LIN {X 0,Y 269.087,Z 444.894,A -85,B 0,C 180,E1 -18604.681,E2 -18604.681} C_VEL
LIN {X 0,Y 267.627,Z 456.093,A -85,B 0,C 180,E1 -18605.777,E2 -18605.777} C_VEL
LIN {X 0,Y 265.719,Z 467.668,A -85,B 0,C 180,E1 -18607.245,E2 -18607.245} C_VEL
LIN {X 0,Y 263.911,Z 478.137,A -85,B 0,C 180,E1 -18608.962,E2 -18608.962} C_VEL
LIN {X 0,Y 262.001,Z 487.303,A -85,B 0,C 180,E1 -18610.818,E2 -18610.818} C_VEL
LIN {X 0,Y 259.893,Z 496.269,A -85,B 0,C 180,E1 -18613.102,E2 -18613.102} C_VEL
LIN {X 0,Y 258.271,Z 503.459,A -85,B 0,C 180,E1 -18615.423,E2 -18615.423} C_VEL
LIN {X 0,Y 256.682,Z 510.056,A -85,B 0,C 180,E1 -18618.152,E2 -18618.152} C_VEL
LIN {X 0,Y 255.709,Z 514.379,A -85,B 0,C 180,E1 -18620.51,E2 -18620.51} C_VEL
LIN {X 0,Y 255.059,Z 517.472,A -85,B 0,C 180,E1 -18622.731,E2 -18622.731} C_VEL
LIN {X 0,Y 254.598,Z 519.914,A -85,B 0,C 180,E1 -18625.251,E2 -18625.251} C_VEL
LIN {X 0,Y 254.212,Z 521.518,A -85,B 0,C 180,E1 -18628.417,E2 -18628.417} C_VEL
LIN {X 0,Y 254.18,Z 521.749,A -85,B 0,C 180,E1 -18630.002,E2 -18630.002} C_VEL
LIN {X 0,Y 254.364,Z 520.966,A -85,B 0,C 180,E1 -18633.169,E2 -18633.169} C_VEL
LIN {X 0,Y 254.595,Z 519.999,A -85,B 0,C 180,E1 -18634.752,E2 -18634.752} C_VEL
LIN {X 0,Y 255.074,Z 517.58,A -85,B 0,C 180,E1 -18637.295,E2 -18637.295} C_VEL
LIN {X 0,Y 255.634,Z 514.567,A -85,B 0,C 180,E1 -18639.496,E2 -18639.496} C_VEL
LIN {X 0,Y 256.622,Z 510.299,A -85,B 0,C 180,E1 -18641.854,E2 -18641.854} C_VEL
LIN {X 0,Y 257.962,Z 504.844,A -85,B 0,C 180,E1 -18644.195,E2 -18644.195} C_VEL
LIN {X 0,Y 259.535,Z 497.997,A -85,B 0,C 180,E1 -18646.52,E2 -18646.52} C_VEL
LIN {X 0,Y 261.635,Z 489.404,A -85,B 0,C 180,E1 -18648.806,E2 -18648.806} C_VEL
LIN {X 0,Y 263.444,Z 480.947,A -85,B 0,C 180,E1 -18650.627,E2 -18650.627} C_VEL
LIN {X 0,Y 265.212,Z 470.915,A -85,B 0,C 180,E1 -18652.393,E2 -18652.393} C_VEL
LIN {X 0,Y 267.064,Z 460.167,A -85,B 0,C 180,E1 -18653.868,E2 -18653.868} C_VEL
LIN {X 0,Y 268.762,Z 448.198,A -85,B 0,C 180,E1 -18655.148,E2 -18655.148} C_VEL
LIN {X 0,Y 270.109,Z 435.553,A -85,B 0,C 180,E1 -18656.15,E2 -18656.15} C_VEL
LIN {X 0,Y 271.18,Z 422.049,A -85,B 0,C 180,E1 -18656.868,E2 -18656.868} C_VEL
LIN {X 0,Y 271.846,Z 405.573,A -85,B 0,C 180,E1 -18657.369,E2 -18657.369} C_VEL
LIN {X 0,Y 273.565,Z 348.69,A -85,B 0,C 180,E1 -18658.847,E2 -18658.847} C_VEL
LIN {X 0,Y 265.912,Z 332.327,A -85,B 0,C 180,E1 -18660.269,E2 -18660.269} C_VEL
LIN {X 0,Y 257.649,Z 317.178,A -85,B 0,C 180,E1 -18661.844,E2 -18661.844} C_VEL
LIN {X 0,Y 256.315,Z 314.678,A -85,B 0,C 180,E1 -18662.112,E2 -18662.112} C_VEL
LIN {X 0,Y 256.105,Z 313.584,A -85,B 0,C 180,E1 -18662.211,E2 -18662.211} C_VEL
LIN {X 0,Y 256.126,Z 313.582,A -85,B 0,C 180,E1 -18665.188,E2 -18665.188} C_VEL
LIN {X 0,Y 256.097,Z 313.587,A -85,B 0,C 180,E1 -18669.139,E2 -18669.139} C_VEL
LIN {X 0,Y 256.078,Z 313.582,A -85,B 0,C 180,E1 -18673.326,E2 -18673.326} C_VEL
LIN {X 0,Y 256.079,Z 313.572,A -85,B 0,C 180,E1 -18677.819,E2 -18677.819} C_VEL
LIN {X 0,Y 256.077,Z 313.589,A -85,B 0,C 180,E1 -18680.859,E2 -18680.859} C_VEL
LIN {X 0,Y 256.135,Z 313.573,A -85,B 0,C 180,E1 -18682.868,E2 -18682.868} C_VEL
LIN {X 0,Y 256.073,Z 313.588,A -85,B 0,C 180,E1 -18686.708,E2 -18686.708} C_VEL
LIN {X 0,Y 256.119,Z 313.574,A -85,B 0,C 180,E1 -18690.401,E2 -18690.401} C_VEL
LIN {X 0,Y 256.217,Z 313.561,A -85,B 0,C 180,E1 -18694.995,E2 -18694.995} C_VEL
LIN {X 0,Y 263.531,Z 341.555,A -85,B 0,C 180,E1 -18696.573,E2 -18696.573} C_VEL
LIN {X 0,Y 260.281,Z 420.849,A -85,B 0,C 180,E1 -18700.068,E2 -18700.068} C_VEL
LIN {X 0,Y 260.015,Z 427.794,A -85,B 0,C 180,E1 -18700.495,E2 -18700.495} C_VEL
LIN {X 0,Y 258.964,Z 433.354,A -85,B 0,C 180,E1 -18700.879,E2 -18700.879} C_VEL
LIN {X 0,Y 255.487,Z 442.099,A -85,B 0,C 180,E1 -18701.589,E2 -18701.589} C_VEL
LIN {X 0,Y 252.06,Z 450.609,A -85,B 0,C 180,E1 -18702.446,E2 -18702.446} C_VEL
LIN {X 0,Y 251.094,Z 455.788,A -85,B 0,C 180,E1 -18703.062,E2 -18703.062} C_VEL
LIN {X 0,Y 250.361,Z 465.042,A -85,B 0,C 180,E1 -18704.324,E2 -18704.324} C_VEL
LIN {X 0,Y 249.484,Z 476.008,A -85,B 0,C 180,E1 -18706.146,E2 -18706.146} C_VEL
LIN {X 0,Y 248.674,Z 486,A -85,B 0,C 180,E1 -18708.176,E2 -18708.176} C_VEL
LIN {X 0,Y 248.087,Z 494.293,A -85,B 0,C 180,E1 -18710.214,E2 -18710.214} C_VEL
LIN {X 0,Y 247.557,Z 502.409,A -85,B 0,C 180,E1 -18712.66,E2 -18712.66} C_VEL
LIN {X 0,Y 247.21,Z 508.939,A -85,B 0,C 180,E1 -18715.107,E2 -18715.107} C_VEL
LIN {X 0,Y 247.148,Z 514.155,A -85,B 0,C 180,E1 -18717.555,E2 -18717.555} C_VEL
LIN {X 0,Y 247.07,Z 518.167,A -85,B 0,C 180,E1 -18720,E2 -18720} C_VEL
LIN {X 0,Y 247.189,Z 520.272,A -85,B 0,C 180,E1 -18721.629,E2 -18721.629} C_VEL
LIN {X 0,Y 247.43,Z 521.895,A -85,B 0,C 180,E1 -18723.257,E2 -18723.257} C_VEL
LIN {X 0,Y 247.715,Z 523.106,A -85,B 0,C 180,E1 -18724.883,E2 -18724.883} C_VEL
LIN {X 0,Y 248.077,Z 523.926,A -85,B 0,C 180,E1 -18726.507,E2 -18726.507} C_VEL
LIN {X 0,Y 249.255,Z 524.369,A -85,B 0,C 180,E1 -18729.29,E2 -18729.29} C_VEL
LIN {X 0,Y 250.523,Z 523.882,A -85,B 0,C 180,E1 -18731.325,E2 -18731.325} C_VEL
LIN {X 0,Y 252.837,Z 521.893,A -85,B 0,C 180,E1 -18734.487,E2 -18734.487} C_VEL
LIN {X 0,Y 255.28,Z 519.262,A -85,B 0,C 180,E1 -18736.802,E2 -18736.802} C_VEL
LIN {X 0,Y 258.013,Z 515.67,A -85,B 0,C 180,E1 -18739.079,E2 -18739.079} C_VEL
LIN {X 0,Y 261.191,Z 511.028,A -85,B 0,C 180,E1 -18741.3,E2 -18741.3} C_VEL
LIN {X 0,Y 265.442,Z 504.122,A -85,B 0,C 180,E1 -18743.814,E2 -18743.814} C_VEL
LIN {X 0,Y 270.342,Z 495.356,A -85,B 0,C 180,E1 -18746.228,E2 -18746.228} C_VEL
LIN {X 0,Y 274.943,Z 485.994,A -85,B 0,C 180,E1 -18748.222,E2 -18748.222} C_VEL
LIN {X 0,Y 279.433,Z 475.658,A -85,B 0,C 180,E1 -18749.992,E2 -18749.992} C_VEL
LIN {X 0,Y 283.883,Z 464.048,A -85,B 0,C 180,E1 -18751.533,E2 -18751.533} C_VEL
LIN {X 0,Y 288.003,Z 451.271,A -85,B 0,C 180,E1 -18752.885,E2 -18752.885} C_VEL
LIN {X 0,Y 291.73,Z 437.57,A -85,B 0,C 180,E1 -18753.959,E2 -18753.959} C_VEL
LIN {X 0,Y 294.428,Z 424.942,A -85,B 0,C 180,E1 -18754.691,E2 -18754.691} C_VEL
LIN {X 0,Y 301.418,Z 387.209,A -85,B 0,C 180,E1 -18756.436,E2 -18756.436} C_VEL
LIN {X 0,Y 299.691,Z 383.358,A -85,B 0,C 180,E1 -18758.133,E2 -18758.133} C_VEL
LIN {X 0,Y 298.164,Z 380.681,A -85,B 0,C 180,E1 -18759.997,E2 -18759.997} C_VEL
LIN {X 0,Y 296.756,Z 378.932,A -85,B 0,C 180,E1 -18762.762,E2 -18762.762} C_VEL
LIN {X 0,Y 296.466,Z 379.001,A -85,B 0,C 180,E1 -18764.984,E2 -18764.984} C_VEL
LIN {X 0,Y 296.557,Z 380.147,A -85,B 0,C 180,E1 -18766.453,E2 -18766.453} C_VEL
LIN {X 0,Y 297.703,Z 384.492,A -85,B 0,C 180,E1 -18769.469,E2 -18769.469} C_VEL
LIN {X 0,Y 299.157,Z 389.614,A -85,B 0,C 180,E1 -18771.566,E2 -18771.566} C_VEL
LIN {X 0,Y 300.305,Z 394.278,A -85,B 0,C 180,E1 -18772.933,E2 -18772.933} C_VEL
LIN {X 0,Y 300.019,Z 397.921,A -85,B 0,C 180,E1 -18773.303,E2 -18773.303} C_VEL
LIN {X 0,Y 292.072,Z 440.822,A -85,B 0,C 180,E1 -18775.25,E2 -18775.25} C_VEL
LIN {X 0,Y 288.407,Z 455.283,A -85,B 0,C 180,E1 -18776.121,E2 -18776.121} C_VEL
LIN {X 0,Y 284.066,Z 469.15,A -85,B 0,C 180,E1 -18777.233,E2 -18777.233} C_VEL
LIN {X 0,Y 279.463,Z 481.671,A -85,B 0,C 180,E1 -18778.544,E2 -18778.544} C_VEL
LIN {X 0,Y 274.353,Z 494.035,A -85,B 0,C 180,E1 -18780.242,E2 -18780.242} C_VEL
LIN {X 0,Y 269.677,Z 504.242,A -85,B 0,C 180,E1 -18782.023,E2 -18782.023} C_VEL
LIN {X 0,Y 265.145,Z 513.442,A -85,B 0,C 180,E1 -18784.063,E2 -18784.063} C_VEL
LIN {X 0,Y 261.091,Z 521.078,A -85,B 0,C 180,E1 -18786.185,E2 -18786.185} C_VEL
LIN {X 0,Y 257.423,Z 527.418,A -85,B 0,C 180,E1 -18788.367,E2 -18788.367} C_VEL
LIN {X 0,Y 254.576,Z 532.571,A -85,B 0,C 180,E1 -18790.652,E2 -18790.652} C_VEL
LIN {X 0,Y 252.113,Z 536.709,A -85,B 0,C 180,E1 -18792.979,E2 -18792.979} C_VEL
LIN {X 0,Y 250.025,Z 539.89,A -85,B 0,C 180,E1 -18795.344,E2 -18795.344} C_VEL
LIN {X 0,Y 248.241,Z 542.675,A -85,B 0,C 180,E1 -18798.568,E2 -18798.568} C_VEL
LIN {X 0,Y 247.251,Z 543.919,A -85,B 0,C 180,E1 -18801.828,E2 -18801.828} C_VEL
LIN {X 0,Y 247.04,Z 543.519,A -85,B 0,C 180,E1 -18805.102,E2 -18805.102} C_VEL
LIN {X 0,Y 247.072,Z 543.112,A -85,B 0,C 180,E1 -18806.357,E2 -18806.357} C_VEL
LIN {X 0,Y 247.095,Z 543.924,A -85,B 0,C 180,E1 -18808.369,E2 -18808.369} C_VEL
LIN {X 0,Y 247.224,Z 544.148,A -85,B 0,C 180,E1 -18809.998,E2 -18809.998} C_VEL
LIN {X 0,Y 247.139,Z 543.916,A -85,B 0,C 180,E1 -18811.628,E2 -18811.628} C_VEL
LIN {X 0,Y 247.041,Z 543.284,A -85,B 0,C 180,E1 -18813.26,E2 -18813.26} C_VEL
LIN {X 0,Y 246.951,Z 542.125,A -85,B 0,C 180,E1 -18815.08,E2 -18815.08} C_VEL
LIN {X 0,Y 247.192,Z 538.891,A -85,B 0,C 180,E1 -18818.171,E2 -18818.171} C_VEL
LIN {X 0,Y 247.681,Z 535.184,A -85,B 0,C 180,E1 -18820.627,E2 -18820.627} C_VEL
LIN {X 0,Y 248.483,Z 530.34,A -85,B 0,C 180,E1 -18823.076,E2 -18823.076} C_VEL
LIN {X 0,Y 249.928,Z 524.229,A -85,B 0,C 180,E1 -18825.492,E2 -18825.492} C_VEL
LIN {X 0,Y 251.653,Z 516.619,A -85,B 0,C 180,E1 -18827.889,E2 -18827.889} C_VEL
LIN {X 0,Y 253.266,Z 508.806,A -85,B 0,C 180,E1 -18829.871,E2 -18829.871} C_VEL
LIN {X 0,Y 255.341,Z 499.264,A -85,B 0,C 180,E1 -18831.811,E2 -18831.811} C_VEL
LIN {X 0,Y 257.545,Z 488.681,A -85,B 0,C 180,E1 -18833.52,E2 -18833.52} C_VEL
LIN {X 0,Y 259.374,Z 478.44,A -85,B 0,C 180,E1 -18834.832,E2 -18834.832} C_VEL
LIN {X 0,Y 261.082,Z 467.279,A -85,B 0,C 180,E1 -18835.938,E2 -18835.938} C_VEL
LIN {X 0,Y 262.693,Z 454.054,A -85,B 0,C 180,E1 -18836.89,E2 -18836.89} C_VEL
LIN {X 0,Y 263.806,Z 441.539,A -85,B 0,C 180,E1 -18837.483,E2 -18837.483} C_VEL
LIN {X 0,Y 265.629,Z 384.766,A -85,B 0,C 180,E1 -18839.024,E2 -18839.024} C_VEL
LIN {X 0,Y 261.716,Z 352.974,A -85,B 0,C 180,E1 -18840.477,E2 -18840.477} C_VEL
LIN {X 0,Y 260.479,Z 344.507,A -85,B 0,C 180,E1 -18840.9,E2 -18840.9} C_VEL
LIN {X 0,Y 253.85,Z 326.102,A -85,B 0,C 180,E1 -18842.391,E2 -18842.391} C_VEL
LIN {X 0,Y 250.812,Z 318.273,A -85,B 0,C 180,E1 -18843.122,E2 -18843.122} C_VEL
LIN {X 0,Y 249.277,Z 315.423,A -85,B 0,C 180,E1 -18843.494,E2 -18843.494} C_VEL
LIN {X 0,Y 249.094,Z 314.457,A -85,B 0,C 180,E1 -18843.611,E2 -18843.611} C_VEL
LIN {X 0,Y 249.044,Z 314.46,A -85,B 0,C 180,E1 -18847.8,E2 -18847.8} C_VEL
LIN {X 0,Y 249.001,Z 314.464,A -85,B 0,C 180,E1 -18850.477,E2 -18850.477} C_VEL
LIN {X 0,Y 248.978,Z 314.467,A -85,B 0,C 180,E1 -18854.882,E2 -18854.882} C_VEL
LIN {X 0,Y 248.978,Z 314.462,A -85,B 0,C 180,E1 -18857.355,E2 -18857.355} C_VEL
LIN {X 0,Y 249.014,Z 314.464,A -85,B 0,C 180,E1 -18862.206,E2 -18862.206} C_VEL
LIN {X 0,Y 249.035,Z 314.458,A -85,B 0,C 180,E1 -18865.638,E2 -18865.638} C_VEL
LIN {X 0,Y 248.986,Z 314.465,A -85,B 0,C 180,E1 -18869.464,E2 -18869.464} C_VEL
LIN {X 0,Y 249.007,Z 314.468,A -85,B 0,C 180,E1 -18873.155,E2 -18873.155} C_VEL
LIN {X 0,Y 249.003,Z 314.466,A -85,B 0,C 180,E1 -18876.725,E2 -18876.725} C_VEL
LIN {X 0,Y 249.05,Z 314.449,A -85,B 0,C 180,E1 -18880.207,E2 -18880.207} C_VEL
LIN {X 0,Y 249.15,Z 314.421,A -85,B 0,C 180,E1 -18883.616,E2 -18883.616} C_VEL
LIN {X 0,Y 249.203,Z 314.439,A -85,B 0,C 180,E1 -18886.961,E2 -18886.961} C_VEL
LIN {X 0,Y 249.375,Z 314.415,A -85,B 0,C 180,E1 -18890.522,E2 -18890.522} C_VEL
LIN {X 0,Y 249.416,Z 314.38,A -85,B 0,C 180,E1 -18893.528,E2 -18893.528} C_VEL
LIN {X 0,Y 249.649,Z 314.38,A -85,B 0,C 180,E1 -18898.387,E2 -18898.387} C_VEL
LIN {X 0,Y 249.65,Z 314.383,A -85,B 0,C 180,E1 -18901.613,E2 -18901.613} C_VEL
LIN {X 0,Y 249.405,Z 314.415,A -85,B 0,C 180,E1 -18906.662,E2 -18906.662} C_VEL
LIN {X 0,Y 249.335,Z 314.417,A -85,B 0,C 180,E1 -18909.737,E2 -18909.737} C_VEL
LIN {X 0,Y 249.168,Z 314.443,A -85,B 0,C 180,E1 -18914.706,E2 -18914.706} C_VEL
LIN {X 0,Y 249.101,Z 314.443,A -85,B 0,C 180,E1 -18918.08,E2 -18918.08} C_VEL
LIN {X 0,Y 249.073,Z 314.458,A -85,B 0,C 180,E1 -18921.52,E2 -18921.52} C_VEL
LIN {X 0,Y 249.097,Z 314.444,A -85,B 0,C 180,E1 -18925.47,E2 -18925.47} C_VEL
LIN {X 0,Y 249.034,Z 314.464,A -85,B 0,C 180,E1 -18928.977,E2 -18928.977} C_VEL
LIN {X 0,Y 249.021,Z 314.454,A -85,B 0,C 180,E1 -18932.427,E2 -18932.427} C_VEL
LIN {X 0,Y 249.042,Z 314.46,A -85,B 0,C 180,E1 -18936.344,E2 -18936.344} C_VEL
LIN {X 0,Y 249.001,Z 314.47,A -85,B 0,C 180,E1 -18940.479,E2 -18940.479} C_VEL
LIN {X 0,Y 248.989,Z 314.471,A -85,B 0,C 180,E1 -18944.883,E2 -18944.883} C_VEL
LIN {X 0,Y 249.012,Z 314.459,A -85,B 0,C 180,E1 -18947.364,E2 -18947.364} C_VEL
LIN {X 0,Y 249.041,Z 314.443,A -85,B 0,C 180,E1 -18952.202,E2 -18952.202} C_VEL
LIN {X 0,Y 249.054,Z 314.462,A -85,B 0,C 180,E1 -18955.643,E2 -18955.643} C_VEL
LIN {X 0,Y 249.043,Z 314.455,A -85,B 0,C 180,E1 -18956.913,E2 -18956.913} C_VEL
LIN {X 0,Y 250.179,Z 317.525,A -85,B 0,C 180,E1 -18957.232,E2 -18957.232} C_VEL
LIN {X 0,Y 255.198,Z 326.145,A -85,B 0,C 180,E1 -18958.242,E2 -18958.242} C_VEL
LIN {X 0,Y 263.451,Z 342.159,A -85,B 0,C 180,E1 -18959.855,E2 -18959.855} C_VEL
LIN {X 0,Y 267.251,Z 350.558,A -85,B 0,C 180,E1 -18960.587,E2 -18960.587} C_VEL
LIN {X 0,Y 264.927,Z 419.914,A -85,B 0,C 180,E1 -18962.464,E2 -18962.464} C_VEL
LIN {X 0,Y 263.995,Z 432.708,A -85,B 0,C 180,E1 -18963.093,E2 -18963.093} C_VEL
LIN {X 0,Y 262.699,Z 445.193,A -85,B 0,C 180,E1 -18964.02,E2 -18964.02} C_VEL
LIN {X 0,Y 261.185,Z 456.398,A -85,B 0,C 180,E1 -18965.14,E2 -18965.14} C_VEL
LIN {X 0,Y 259.426,Z 466.702,A -85,B 0,C 180,E1 -18966.45,E2 -18966.45} C_VEL
LIN {X 0,Y 257.635,Z 476.588,A -85,B 0,C 180,E1 -18968.046,E2 -18968.046} C_VEL
LIN {X 0,Y 255.736,Z 485.882,A -85,B 0,C 180,E1 -18969.91,E2 -18969.91} C_VEL
LIN {X 0,Y 253.438,Z 495.252,A -85,B 0,C 180,E1 -18972.241,E2 -18972.241} C_VEL
LIN {X 0,Y 251.682,Z 502.686,A -85,B 0,C 180,E1 -18974.618,E2 -18974.618} C_VEL
LIN {X 0,Y 250.172,Z 508.656,A -85,B 0,C 180,E1 -18977.014,E2 -18977.014} C_VEL
LIN {X 0,Y 249.021,Z 513.369,A -85,B 0,C 180,E1 -18979.431,E2 -18979.431} C_VEL
LIN {X 0,Y 248.22,Z 516.967,A -85,B 0,C 180,E1 -18981.863,E2 -18981.863} C_VEL
LIN {X 0,Y 247.791,Z 518.82,A -85,B 0,C 180,E1 -18983.487,E2 -18983.487} C_VEL
LIN {X 0,Y 247.531,Z 520.231,A -85,B 0,C 180,E1 -18985.115,E2 -18985.115} C_VEL
LIN {X 0,Y 247.305,Z 521.222,A -85,B 0,C 180,E1 -18986.743,E2 -18986.743} C_VEL
LIN {X 0,Y 247.105,Z 522.065,A -85,B 0,C 180,E1 -18990.002,E2 -18990.002} C_VEL
LIN {X 0,Y 247.304,Z 521.282,A -85,B 0,C 180,E1 -18993.26,E2 -18993.26} C_VEL
LIN {X 0,Y 247.528,Z 520.315,A -85,B 0,C 180,E1 -18994.888,E2 -18994.888} C_VEL
LIN {X 0,Y 248.006,Z 518.084,A -85,B 0,C 180,E1 -18997.327,E2 -18997.327} C_VEL
LIN {X 0,Y 248.648,Z 514.882,A -85,B 0,C 180,E1 -18999.766,E2 -18999.766} C_VEL
LIN {X 0,Y 249.691,Z 510.613,A -85,B 0,C 180,E1 -19002.188,E2 -19002.188} C_VEL
LIN {X 0,Y 251.08,Z 505.157,A -85,B 0,C 180,E1 -19004.593,E2 -19004.593} C_VEL
LIN {X 0,Y 252.742,Z 498.308,A -85,B 0,C 180,E1 -19006.978,E2 -19006.978} C_VEL
LIN {X 0,Y 254.939,Z 489.713,A -85,B 0,C 180,E1 -19009.319,E2 -19009.319} C_VEL
LIN {X 0,Y 257.036,Z 480.126,A -85,B 0,C 180,E1 -19011.414,E2 -19011.414} C_VEL
LIN {X 0,Y 258.928,Z 469.969,A -85,B 0,C 180,E1 -19013.178,E2 -19013.178} C_VEL
LIN {X 0,Y 260.859,Z 458.939,A -85,B 0,C 180,E1 -19014.684,E2 -19014.684} C_VEL
LIN {X 0,Y 262.494,Z 447.523,A -85,B 0,C 180,E1 -19015.898,E2 -19015.898} C_VEL
LIN {X 0,Y 263.836,Z 435.113,A -85,B 0,C 180,E1 -19016.874,E2 -19016.874} C_VEL
LIN {X 0,Y 264.925,Z 421.576,A -85,B 0,C 180,E1 -19017.593,E2 -19017.593} C_VEL
LIN {X 0,Y 265.871,Z 399.693,A -85,B 0,C 180,E1 -19018.22,E2 -19018.22} C_VEL
LIN {X 0,Y 267.382,Z 350.81,A -85,B 0,C 180,E1 -19019.521,E2 -19019.521} C_VEL
LIN {X 0,Y 260.253,Z 335.662,A -85,B 0,C 180,E1 -19020.899,E2 -19020.899} C_VEL
LIN {X 0,Y 252.615,Z 321.586,A -85,B 0,C 180,E1 -19022.414,E2 -19022.414} C_VEL
LIN {X 0,Y 250.257,Z 317.599,A -85,B 0,C 180,E1 -19022.894,E2 -19022.894} C_VEL
LIN {X 0,Y 249.241,Z 315.427,A -85,B 0,C 180,E1 -19023.12,E2 -19023.12} C_VEL
LIN {X 0,Y 249.062,Z 314.462,A -85,B 0,C 180,E1 -19023.214,E2 -19023.214} C_VEL
LIN {X 0,Y 249.074,Z 314.457,A -85,B 0,C 180,E1 -19026.34,E2 -19026.34} C_VEL
LIN {X 0,Y 249.037,Z 314.465,A -85,B 0,C 180,E1 -19030.474,E2 -19030.474} C_VEL
LIN {X 0,Y 249.015,Z 314.441,A -85,B 0,C 180,E1 -19034.878,E2 -19034.878} C_VEL
LIN {X 0,Y 249.024,Z 314.443,A -85,B 0,C 180,E1 -19037.364,E2 -19037.364} C_VEL
LIN {X 0,Y 249.049,Z 314.459,A -85,B 0,C 180,E1 -19042.201,E2 -19042.201} C_VEL
LIN {X 0,Y 249.049,Z 314.462,A -85,B 0,C 180,E1 -19045.64,E2 -19045.64} C_VEL
LIN {X 0,Y 249.057,Z 314.45,A -85,B 0,C 180,E1 -19049.474,E2 -19049.474} C_VEL
LIN {X 0,Y 249.085,Z 314.457,A -85,B 0,C 180,E1 -19053.163,E2 -19053.163} C_VEL
LIN {X 0,Y 249.16,Z 314.441,A -85,B 0,C 180,E1 -19054.746,E2 -19054.746} C_VEL
LIN {X 0,Y 256.508,Z 342.412,A -85,B 0,C 180,E1 -19056.356,E2 -19056.356} C_VEL
LIN {X 0,Y 253.206,Z 421.109,A -85,B 0,C 180,E1 -19059.964,E2 -19059.964} C_VEL
LIN {X 0,Y 252.526,Z 433.681,A -85,B 0,C 180,E1 -19060.822,E2 -19060.822} C_VEL
LIN {X 0,Y 251.809,Z 445.98,A -85,B 0,C 180,E1 -19061.941,E2 -19061.941} C_VEL
LIN {X 0,Y 251.094,Z 455.788,A -85,B 0,C 180,E1 -19063.062,E2 -19063.062} C_VEL
LIN {X 0,Y 250.112,Z 460.857,A -85,B 0,C 180,E1 -19063.717,E2 -19063.717} C_VEL
LIN {X 0,Y 246.62,Z 468.667,A -85,B 0,C 180,E1 -19064.875,E2 -19064.875} C_VEL
LIN {X 0,Y 243.057,Z 476.081,A -85,B 0,C 180,E1 -19066.196,E2 -19066.196} C_VEL
LIN {X 0,Y 241.982,Z 480.538,A -85,B 0,C 180,E1 -19067.089,E2 -19067.089} C_VEL
LIN {X 0,Y 241.188,Z 491.086,A -85,B 0,C 180,E1 -19069.507,E2 -19069.507} C_VEL
LIN {X 0,Y 240.585,Z 499.864,A -85,B 0,C 180,E1 -19072.024,E2 -19072.024} C_VEL
LIN {X 0,Y 240.207,Z 506.732,A -85,B 0,C 180,E1 -19074.444,E2 -19074.444} C_VEL
LIN {X 0,Y 240.163,Z 511.814,A -85,B 0,C 180,E1 -19076.645,E2 -19076.645} C_VEL
LIN {X 0,Y 239.984,Z 516.456,A -85,B 0,C 180,E1 -19079.161,E2 -19079.161} C_VEL
LIN {X 0,Y 240.12,Z 519.99,A -85,B 0,C 180,E1 -19081.677,E2 -19081.677} C_VEL
LIN {X 0,Y 240.347,Z 521.802,A -85,B 0,C 180,E1 -19083.353,E2 -19083.353} C_VEL
LIN {X 0,Y 240.65,Z 523.175,A -85,B 0,C 180,E1 -19085.026,E2 -19085.026} C_VEL
LIN {X 0,Y 241.655,Z 524.669,A -85,B 0,C 180,E1 -19088.361,E2 -19088.361} C_VEL
LIN {X 0,Y 242.528,Z 524.83,A -85,B 0,C 180,E1 -19090.013,E2 -19090.013} C_VEL
LIN {X 0,Y 243.608,Z 524.588,A -85,B 0,C 180,E1 -19091.651,E2 -19091.651} C_VEL
LIN {X 0,Y 246.066,Z 522.889,A -85,B 0,C 180,E1 -19094.895,E2 -19094.895} C_VEL
LIN {X 0,Y 249.518,Z 519.587,A -85,B 0,C 180,E1 -19098.049,E2 -19098.049} C_VEL
LIN {X 0,Y 252.569,Z 515.969,A -85,B 0,C 180,E1 -19100.354,E2 -19100.354} C_VEL
LIN {X 0,Y 256.035,Z 511.318,A -85,B 0,C 180,E1 -19102.6,E2 -19102.6} C_VEL
LIN {X 0,Y 260.666,Z 504.393,A -85,B 0,C 180,E1 -19105.128,E2 -19105.128} C_VEL
LIN {X 0,Y 265.948,Z 495.64,A -85,B 0,C 180,E1 -19107.546,E2 -19107.546} C_VEL
LIN {X 0,Y 270.882,Z 486.311,A -85,B 0,C 180,E1 -19109.535,E2 -19109.535} C_VEL
LIN {X 0,Y 275.658,Z 476.045,A -85,B 0,C 180,E1 -19111.297,E2 -19111.297} C_VEL
LIN {X 0,Y 280.844,Z 463.286,A -85,B 0,C 180,E1 -19112.976,E2 -19112.976} C_VEL
LIN {X 0,Y 284.759,Z 451.85,A -85,B 0,C 180,E1 -19114.158,E2 -19114.158} C_VEL
LIN {X 0,Y 288.683,Z 438.403,A -85,B 0,C 180,E1 -19115.217,E2 -19115.217} C_VEL
LIN {X 0,Y 291.853,Z 424.432,A -85,B 0,C 180,E1 -19116.024,E2 -19116.024} C_VEL
LIN {X 0,Y 298.24,Z 392.213,A -85,B 0,C 180,E1 -19117.49,E2 -19117.49} C_VEL
LIN {X 0,Y 298.184,Z 391.567,A -85,B 0,C 180,E1 -19117.638,E2 -19117.638} C_VEL
LIN {X 0,Y 297.122,Z 389.363,A -85,B 0,C 180,E1 -19118.827,E2 -19118.827} C_VEL
LIN {X 0,Y 296.061,Z 387.308,A -85,B 0,C 180,E1 -19120.347,E2 -19120.347} C_VEL
LIN {X 0,Y 294.865,Z 385.71,A -85,B 0,C 180,E1 -19123.04,E2 -19123.04} C_VEL
LIN {X 0,Y 294.641,Z 386.057,A -85,B 0,C 180,E1 -19125.349,E2 -19125.349} C_VEL
LIN {X 0,Y 294.894,Z 388.583,A -85,B 0,C 180,E1 -19127.533,E2 -19127.533} C_VEL
LIN {X 0,Y 295.797,Z 391.92,A -85,B 0,C 180,E1 -19129.553,E2 -19129.553} C_VEL
LIN {X 0,Y 296.787,Z 396.248,A -85,B 0,C 180,E1 -19131.202,E2 -19131.202} C_VEL
LIN {X 0,Y 297.339,Z 399.057,A -85,B 0,C 180,E1 -19132.026,E2 -19132.026} C_VEL
LIN {X 0,Y 289.411,Z 439.47,A -85,B 0,C 180,E1 -19133.897,E2 -19133.897} C_VEL
LIN {X 0,Y 285.471,Z 454.308,A -85,B 0,C 180,E1 -19134.778,E2 -19134.778} C_VEL
LIN {X 0,Y 281.237,Z 467.257,A -85,B 0,C 180,E1 -19135.786,E2 -19135.786} C_VEL
LIN {X 0,Y 276.407,Z 479.706,A -85,B 0,C 180,E1 -19137.042,E2 -19137.042} C_VEL
LIN {X 0,Y 271.373,Z 491.387,A -85,B 0,C 180,E1 -19138.586,E2 -19138.586} C_VEL
LIN {X 0,Y 266.264,Z 501.845,A -85,B 0,C 180,E1 -19140.335,E2 -19140.335} C_VEL
LIN {X 0,Y 261.278,Z 511.323,A -85,B 0,C 180,E1 -19142.353,E2 -19142.353} C_VEL
LIN {X 0,Y 256.806,Z 519.207,A -85,B 0,C 180,E1 -19144.466,E2 -19144.466} C_VEL
LIN {X 0,Y 252.128,Z 526.704,A -85,B 0,C 180,E1 -19147.029,E2 -19147.029} C_VEL
LIN {X 0,Y 248.895,Z 531.875,A -85,B 0,C 180,E1 -19149.33,E2 -19149.33} C_VEL
LIN {X 0,Y 245.366,Z 537.212,A -85,B 0,C 180,E1 -19152.496,E2 -19152.496} C_VEL
LIN {X 0,Y 243.161,Z 540.098,A -85,B 0,C 180,E1 -19154.921,E2 -19154.921} C_VEL
LIN {X 0,Y 242.078,Z 541.544,A -85,B 0,C 180,E1 -19156.568,E2 -19156.568} C_VEL
LIN {X 0,Y 240.643,Z 543.22,A -85,B 0,C 180,E1 -19159.906,E2 -19159.906} C_VEL
LIN {X 0,Y 240.003,Z 543.355,A -85,B 0,C 180,E1 -19163.272,E2 -19163.272} C_VEL
LIN {X 0,Y 240.007,Z 542.499,A -85,B 0,C 180,E1 -19165.73,E2 -19165.73} C_VEL
LIN {X 0,Y 240.022,Z 543.608,A -85,B 0,C 180,E1 -19168.32,E2 -19168.32} C_VEL
LIN {X 0,Y 240.142,Z 543.832,A -85,B 0,C 180,E1 -19169.998,E2 -19169.998} C_VEL
LIN {X 0,Y 240.06,Z 543.6,A -85,B 0,C 180,E1 -19171.676,E2 -19171.676} C_VEL
LIN {X 0,Y 239.933,Z 542.966,A -85,B 0,C 180,E1 -19173.357,E2 -19173.357} C_VEL
LIN {X 0,Y 239.88,Z 541.939,A -85,B 0,C 180,E1 -19175.041,E2 -19175.041} C_VEL
LIN {X 0,Y 239.949,Z 540.486,A -85,B 0,C 180,E1 -19176.726,E2 -19176.726} C_VEL
LIN {X 0,Y 240.287,Z 537.478,A -85,B 0,C 180,E1 -19179.255,E2 -19179.255} C_VEL
LIN {X 0,Y 240.89,Z 533.403,A -85,B 0,C 180,E1 -19181.782,E2 -19181.782} C_VEL
LIN {X 0,Y 242.241,Z 527.136,A -85,B 0,C 180,E1 -19184.704,E2 -19184.704} C_VEL
LIN {X 0,Y 243.89,Z 520.313,A -85,B 0,C 180,E1 -19187.178,E2 -19187.178} C_VEL
LIN {X 0,Y 245.636,Z 512.779,A -85,B 0,C 180,E1 -19189.371,E2 -19189.371} C_VEL
LIN {X 0,Y 247.365,Z 504.93,A -85,B 0,C 180,E1 -19191.236,E2 -19191.236} C_VEL
LIN {X 0,Y 249.676,Z 494.523,A -85,B 0,C 180,E1 -19193.207,E2 -19193.207} C_VEL
LIN {X 0,Y 252.138,Z 482.81,A -85,B 0,C 180,E1 -19194.933,E2 -19194.933} C_VEL
LIN {X 0,Y 254.071,Z 470.986,A -85,B 0,C 180,E1 -19196.267,E2 -19196.267} C_VEL
LIN {X 0,Y 255.813,Z 458.725,A -85,B 0,C 180,E1 -19197.286,E2 -19197.286} C_VEL
LIN {X 0,Y 257.185,Z 445.828,A -85,B 0,C 180,E1 -19198.022,E2 -19198.022} C_VEL
LIN {X 0,Y 258.01,Z 430.914,A -85,B 0,C 180,E1 -19198.525,E2 -19198.525} C_VEL
LIN {X 0,Y 259.357,Z 385.333,A -85,B 0,C 180,E1 -19199.771,E2 -19199.771} C_VEL
LIN {X 0,Y 255.609,Z 354.011,A -85,B 0,C 180,E1 -19201.245,E2 -19201.245} C_VEL
LIN {X 0,Y 254.553,Z 346.842,A -85,B 0,C 180,E1 -19201.62,E2 -19201.62} C_VEL
LIN {X 0,Y 247.87,Z 328.19,A -85,B 0,C 180,E1 -19203.194,E2 -19203.194} C_VEL
LIN {X 0,Y 245.612,Z 322.502,A -85,B 0,C 180,E1 -19203.731,E2 -19203.731} C_VEL
LIN {X 0,Y 242.331,Z 316.691,A -85,B 0,C 180,E1 -19204.507,E2 -19204.507} C_VEL
LIN {X 0,Y 242.037,Z 315.333,A -85,B 0,C 180,E1 -19204.655,E2 -19204.655} C_VEL
LIN {X 0,Y 241.994,Z 315.341,A -85,B 0,C 180,E1 -19208.359,E2 -19208.359} C_VEL
LIN {X 0,Y 241.929,Z 315.347,A -85,B 0,C 180,E1 -19211.922,E2 -19211.922} C_VEL
LIN {X 0,Y 241.903,Z 315.342,A -85,B 0,C 180,E1 -19216.576,E2 -19216.576} C_VEL
LIN {X 0,Y 241.968,Z 315.337,A -85,B 0,C 180,E1 -19221.645,E2 -19221.645} C_VEL
LIN {X 0,Y 241.966,Z 315.336,A -85,B 0,C 180,E1 -19224.486,E2 -19224.486} C_VEL
LIN {X 0,Y 241.941,Z 315.343,A -85,B 0,C 180,E1 -19228.475,E2 -19228.475} C_VEL
LIN {X 0,Y 241.944,Z 315.346,A -85,B 0,C 180,E1 -19232.305,E2 -19232.305} C_VEL
LIN {X 0,Y 241.977,Z 315.343,A -85,B 0,C 180,E1 -19236.008,E2 -19236.008} C_VEL
LIN {X 0,Y 241.984,Z 315.331,A -85,B 0,C 180,E1 -19239.603,E2 -19239.603} C_VEL
LIN {X 0,Y 242.106,Z 315.294,A -85,B 0,C 180,E1 -19243.317,E2 -19243.317} C_VEL
LIN {X 0,Y 242.142,Z 315.317,A -85,B 0,C 180,E1 -19246.574,E2 -19246.574} C_VEL
LIN {X 0,Y 242.334,Z 315.292,A -85,B 0,C 180,E1 -19250.404,E2 -19250.404} C_VEL
LIN {X 0,Y 242.387,Z 315.254,A -85,B 0,C 180,E1 -19253.34,E2 -19253.34} C_VEL
LIN {X 0,Y 242.609,Z 315.257,A -85,B 0,C 180,E1 -19258.34,E2 -19258.34} C_VEL
LIN {X 0,Y 242.61,Z 315.259,A -85,B 0,C 180,E1 -19261.66,E2 -19261.66} C_VEL
LIN {X 0,Y 242.387,Z 315.292,A -85,B 0,C 180,E1 -19266.66,E2 -19266.66} C_VEL
LIN {X 0,Y 242.258,Z 315.298,A -85,B 0,C 180,E1 -19270.024,E2 -19270.024} C_VEL
LIN {X 0,Y 242.127,Z 315.316,A -85,B 0,C 180,E1 -19275.144,E2 -19275.144} C_VEL
LIN {X 0,Y 242.039,Z 315.325,A -85,B 0,C 180,E1 -19278.627,E2 -19278.627} C_VEL
LIN {X 0,Y 241.996,Z 315.34,A -85,B 0,C 180,E1 -19282.182,E2 -19282.182} C_VEL
LIN {X 0,Y 242.025,Z 315.326,A -85,B 0,C 180,E1 -19285.822,E2 -19285.822} C_VEL
LIN {X 0,Y 241.964,Z 315.342,A -85,B 0,C 180,E1 -19289.589,E2 -19289.589} C_VEL
LIN {X 0,Y 241.973,Z 315.339,A -85,B 0,C 180,E1 -19293.494,E2 -19293.494} C_VEL
LIN {X 0,Y 241.983,Z 315.332,A -85,B 0,C 180,E1 -19297.583,E2 -19297.583} C_VEL
LIN {X 0,Y 241.928,Z 315.347,A -85,B 0,C 180,E1 -19301.925,E2 -19301.925} C_VEL
LIN {X 0,Y 241.928,Z 315.345,A -85,B 0,C 180,E1 -19306.573,E2 -19306.573} C_VEL
LIN {X 0,Y 241.953,Z 315.343,A -85,B 0,C 180,E1 -19310.283,E2 -19310.283} C_VEL
LIN {X 0,Y 242.001,Z 315.331,A -85,B 0,C 180,E1 -19314.494,E2 -19314.494} C_VEL
LIN {X 0,Y 241.999,Z 315.342,A -85,B 0,C 180,E1 -19315.86,E2 -19315.86} C_VEL
LIN {X 0,Y 243.079,Z 318.325,A -85,B 0,C 180,E1 -19316.167,E2 -19316.167} C_VEL
LIN {X 0,Y 244.502,Z 320.541,A -85,B 0,C 180,E1 -19316.469,E2 -19316.469} C_VEL
LIN {X 0,Y 253.035,Z 335.811,A -85,B 0,C 180,E1 -19318.254,E2 -19318.254} C_VEL
LIN {X 0,Y 260.05,Z 350.326,A -85,B 0,C 180,E1 -19319.673,E2 -19319.673} C_VEL
LIN {X 0,Y 261.039,Z 352.605,A -85,B 0,C 180,E1 -19319.872,E2 -19319.872} C_VEL
LIN {X 0,Y 258.682,Z 419.682,A -85,B 0,C 180,E1 -19321.72,E2 -19321.72} C_VEL
LIN {X 0,Y 257.753,Z 432.365,A -85,B 0,C 180,E1 -19322.338,E2 -19322.338} C_VEL
LIN {X 0,Y 256.359,Z 445.492,A -85,B 0,C 180,E1 -19323.328,E2 -19323.328} C_VEL
LIN {X 0,Y 254.772,Z 456.703,A -85,B 0,C 180,E1 -19324.469,E2 -19324.469} C_VEL
LIN {X 0,Y 252.956,Z 467.01,A -85,B 0,C 180,E1 -19325.809,E2 -19325.809} C_VEL
LIN {X 0,Y 250.932,Z 477.513,A -85,B 0,C 180,E1 -19327.557,E2 -19327.557} C_VEL
LIN {X 0,Y 249.096,Z 486.195,A -85,B 0,C 180,E1 -19329.351,E2 -19329.351} C_VEL
LIN {X 0,Y 246.699,Z 495.567,A -85,B 0,C 180,E1 -19331.739,E2 -19331.739} C_VEL
LIN {X 0,Y 244.857,Z 503.002,A -85,B 0,C 180,E1 -19334.178,E2 -19334.178} C_VEL
LIN {X 0,Y 243.273,Z 508.972,A -85,B 0,C 180,E1 -19336.639,E2 -19336.639} C_VEL
LIN {X 0,Y 242.049,Z 513.686,A -85,B 0,C 180,E1 -19339.123,E2 -19339.123} C_VEL
LIN {X 0,Y 241.193,Z 517.284,A -85,B 0,C 180,E1 -19341.624,E2 -19341.624} C_VEL
LIN {X 0,Y 240.736,Z 519.138,A -85,B 0,C 180,E1 -19343.296,E2 -19343.296} C_VEL
LIN {X 0,Y 240.467,Z 520.548,A -85,B 0,C 180,E1 -19344.972,E2 -19344.972} C_VEL
LIN {X 0,Y 240.247,Z 521.538,A -85,B 0,C 180,E1 -19346.648,E2 -19346.648} C_VEL
LIN {X 0,Y 240.032,Z 522.381,A -85,B 0,C 180,E1 -19350.002,E2 -19350.002} C_VEL
LIN {X 0,Y 240.246,Z 521.597,A -85,B 0,C 180,E1 -19353.356,E2 -19353.356} C_VEL
LIN {X 0,Y 240.464,Z 520.631,A -85,B 0,C 180,E1 -19355.032,E2 -19355.032} C_VEL
LIN {X 0,Y 240.935,Z 518.595,A -85,B 0,C 180,E1 -19357.354,E2 -19357.354} C_VEL
LIN {X 0,Y 241.659,Z 515.197,A -85,B 0,C 180,E1 -19360.051,E2 -19360.051} C_VEL
LIN {X 0,Y 242.759,Z 510.927,A -85,B 0,C 180,E1 -19362.542,E2 -19362.542} C_VEL
LIN {X 0,Y 244.216,Z 505.471,A -85,B 0,C 180,E1 -19365.012,E2 -19365.012} C_VEL
LIN {X 0,Y 245.974,Z 498.619,A -85,B 0,C 180,E1 -19367.46,E2 -19367.46} C_VEL
LIN {X 0,Y 248.261,Z 490.022,A -85,B 0,C 180,E1 -19369.861,E2 -19369.861} C_VEL
LIN {X 0,Y 250.329,Z 480.955,A -85,B 0,C 180,E1 -19371.9,E2 -19371.9} C_VEL
LIN {X 0,Y 252.434,Z 470.27,A -85,B 0,C 180,E1 -19373.811,E2 -19373.811} C_VEL
LIN {X 0,Y 254.424,Z 459.235,A -85,B 0,C 180,E1 -19375.352,E2 -19375.352} C_VEL
LIN {X 0,Y 256.135,Z 447.811,A -85,B 0,C 180,E1 -19376.591,E2 -19376.591} C_VEL
LIN {X 0,Y 257.552,Z 435.384,A -85,B 0,C 180,E1 -19377.585,E2 -19377.585} C_VEL
LIN {X 0,Y 258.637,Z 422.343,A -85,B 0,C 180,E1 -19378.295,E2 -19378.295} C_VEL
LIN {X 0,Y 259.417,Z 404.989,A -85,B 0,C 180,E1 -19378.829,E2 -19378.829} C_VEL
LIN {X 0,Y 261.102,Z 352.638,A -85,B 0,C 180,E1 -19380.253,E2 -19380.253} C_VEL
LIN {X 0,Y 253.854,Z 337.331,A -85,B 0,C 180,E1 -19381.718,E2 -19381.718} C_VEL
LIN {X 0,Y 245.421,Z 322.148,A -85,B 0,C 180,E1 -19383.475,E2 -19383.475} C_VEL
LIN {X 0,Y 243.343,Z 318.684,A -85,B 0,C 180,E1 -19383.923,E2 -19383.923} C_VEL
LIN {X 0,Y 242.088,Z 315.794,A -85,B 0,C 180,E1 -19384.226,E2 -19384.226} C_VEL
LIN {X 0,Y 242.023,Z 315.338,A -85,B 0,C 180,E1 -19384.258,E2 -19384.258} C_VEL
LIN {X 0,Y 242.014,Z 315.343,A -85,B 0,C 180,E1 -19388.365,E2 -19388.365} C_VEL
LIN {X 0,Y 241.958,Z 315.35,A -85,B 0,C 180,E1 -19391.92,E2 -19391.92} C_VEL
LIN {X 0,Y 241.943,Z 315.317,A -85,B 0,C 180,E1 -19396.571,E2 -19396.571} C_VEL
LIN {X 0,Y 241.962,Z 315.345,A -85,B 0,C 180,E1 -19400.282,E2 -19400.282} C_VEL
LIN {X 0,Y 241.987,Z 315.335,A -85,B 0,C 180,E1 -19404.489,E2 -19404.489} C_VEL
LIN {X 0,Y 241.98,Z 315.334,A -85,B 0,C 180,E1 -19408.48,E2 -19408.48} C_VEL
LIN {X 0,Y 242.017,Z 315.338,A -85,B 0,C 180,E1 -19412.314,E2 -19412.314} C_VEL
LIN {X 0,Y 242.121,Z 315.38,A -85,B 0,C 180,E1 -19414.498,E2 -19414.498} C_VEL
LIN {X 0,Y 249.369,Z 342.598,A -85,B 0,C 180,E1 -19416.107,E2 -19416.107} C_VEL
LIN {X 0,Y 246.127,Z 421.08,A -85,B 0,C 180,E1 -19419.852,E2 -19419.852} C_VEL
LIN {X 0,Y 245.39,Z 434.179,A -85,B 0,C 180,E1 -19420.777,E2 -19420.777} C_VEL
LIN {X 0,Y 244.624,Z 447.112,A -85,B 0,C 180,E1 -19422.01,E2 -19422.01} C_VEL
LIN {X 0,Y 243.73,Z 460.523,A -85,B 0,C 180,E1 -19423.671,E2 -19423.671} C_VEL
LIN {X 0,Y 242.676,Z 472.343,A -85,B 0,C 180,E1 -19425.535,E2 -19425.535} C_VEL
LIN {X 0,Y 241.982,Z 480.538,A -85,B 0,C 180,E1 -19427.089,E2 -19427.089} C_VEL
LIN {X 0,Y 240.94,Z 484.85,A -85,B 0,C 180,E1 -19428.023,E2 -19428.023} C_VEL
LIN {X 0,Y 237.547,Z 491.293,A -85,B 0,C 180,E1 -19429.638,E2 -19429.638} C_VEL
LIN {X 0,Y 234.279,Z 497.291,A -85,B 0,C 180,E1 -19431.404,E2 -19431.404} C_VEL
LIN {X 0,Y 233.447,Z 500.811,A -85,B 0,C 180,E1 -19432.552,E2 -19432.552} C_VEL
LIN {X 0,Y 233.075,Z 508.052,A -85,B 0,C 180,E1 -19435.243,E2 -19435.243} C_VEL
LIN {X 0,Y 233.025,Z 512.742,A -85,B 0,C 180,E1 -19437.407,E2 -19437.407} C_VEL
LIN {X 0,Y 232.929,Z 517.259,A -85,B 0,C 180,E1 -19440,E2 -19440} C_VEL
LIN {X 0,Y 233.052,Z 519.673,A -85,B 0,C 180,E1 -19441.728,E2 -19441.728} C_VEL
LIN {X 0,Y 233.29,Z 521.603,A -85,B 0,C 180,E1 -19443.454,E2 -19443.454} C_VEL
LIN {X 0,Y 233.589,Z 523.13,A -85,B 0,C 180,E1 -19445.179,E2 -19445.179} C_VEL
LIN {X 0,Y 233.983,Z 524.261,A -85,B 0,C 180,E1 -19446.9,E2 -19446.9} C_VEL
LIN {X 0,Y 234.931,Z 525.105,A -85,B 0,C 180,E1 -19449.169,E2 -19449.169} C_VEL
LIN {X 0,Y 236.694,Z 525.188,A -85,B 0,C 180,E1 -19451.996,E2 -19451.996} C_VEL
LIN {X 0,Y 239.301,Z 523.89,A -85,B 0,C 180,E1 -19455.327,E2 -19455.327} C_VEL
LIN {X 0,Y 242.902,Z 520.929,A -85,B 0,C 180,E1 -19458.558,E2 -19458.558} C_VEL
LIN {X 0,Y 247.283,Z 516.339,A -85,B 0,C 180,E1 -19461.683,E2 -19461.683} C_VEL
LIN {X 0,Y 251.064,Z 511.696,A -85,B 0,C 180,E1 -19463.947,E2 -19463.947} C_VEL
LIN {X 0,Y 256.124,Z 504.769,A -85,B 0,C 180,E1 -19466.481,E2 -19466.481} C_VEL
LIN {X 0,Y 261.732,Z 496.089,A -85,B 0,C 180,E1 -19468.903,E2 -19468.903} C_VEL
LIN {X 0,Y 266.994,Z 486.84,A -85,B 0,C 180,E1 -19470.883,E2 -19470.883} C_VEL
LIN {X 0,Y 272.129,Z 476.639,A -85,B 0,C 180,E1 -19472.624,E2 -19472.624} C_VEL
LIN {X 0,Y 277.618,Z 464.036,A -85,B 0,C 180,E1 -19474.282,E2 -19474.282} C_VEL
LIN {X 0,Y 281.746,Z 452.824,A -85,B 0,C 180,E1 -19475.448,E2 -19475.448} C_VEL
LIN {X 0,Y 285.569,Z 440.607,A -85,B 0,C 180,E1 -19476.422,E2 -19476.422} C_VEL
LIN {X 0,Y 288.826,Z 427.842,A -85,B 0,C 180,E1 -19477.195,E2 -19477.195} C_VEL
LIN {X 0,Y 295.378,Z 396.767,A -85,B 0,C 180,E1 -19478.617,E2 -19478.617} C_VEL
LIN {X 0,Y 294.083,Z 394.075,A -85,B 0,C 180,E1 -19480.508,E2 -19480.508} C_VEL
LIN {X 0,Y 292.986,Z 392.538,A -85,B 0,C 180,E1 -19483.217,E2 -19483.217} C_VEL
LIN {X 0,Y 292.799,Z 392.93,A -85,B 0,C 180,E1 -19485.335,E2 -19485.335} C_VEL
LIN {X 0,Y 293.104,Z 396.269,A -85,B 0,C 180,E1 -19487.912,E2 -19487.912} C_VEL
LIN {X 0,Y 293.607,Z 398.346,A -85,B 0,C 180,E1 -19489.121,E2 -19489.121} C_VEL
LIN {X 0,Y 294.387,Z 402.455,A -85,B 0,C 180,E1 -19490.715,E2 -19490.715} C_VEL
LIN {X 0,Y 294.459,Z 403.166,A -85,B 0,C 180,E1 -19490.901,E2 -19490.901} C_VEL
LIN {X 0,Y 286.864,Z 439.273,A -85,B 0,C 180,E1 -19492.561,E2 -19492.561} C_VEL
LIN {X 0,Y 282.854,Z 453.507,A -85,B 0,C 180,E1 -19493.392,E2 -19493.392} C_VEL
LIN {X 0,Y 278.072,Z 467.262,A -85,B 0,C 180,E1 -19494.456,E2 -19494.456} C_VEL
LIN {X 0,Y 272.887,Z 479.714,A -85,B 0,C 180,E1 -19495.709,E2 -19495.709} C_VEL
LIN {X 0,Y 268.067,Z 490.195,A -85,B 0,C 180,E1 -19497.086,E2 -19497.086} C_VEL
LIN {X 0,Y 263.202,Z 499.675,A -85,B 0,C 180,E1 -19498.62,E2 -19498.62} C_VEL
LIN {X 0,Y 257.703,Z 509.36,A -85,B 0,C 180,E1 -19500.599,E2 -19500.599} C_VEL
LIN {X 0,Y 252.056,Z 518.638,A -85,B 0,C 180,E1 -19503.056,E2 -19503.056} C_VEL
LIN {X 0,Y 247.04,Z 526.085,A -85,B 0,C 180,E1 -19505.636,E2 -19505.636} C_VEL
LIN {X 0,Y 243.331,Z 531.264,A -85,B 0,C 180,E1 -19507.945,E2 -19507.945} C_VEL
LIN {X 0,Y 239.464,Z 536.587,A -85,B 0,C 180,E1 -19511.164,E2 -19511.164} C_VEL
LIN {X 0,Y 237.766,Z 538.642,A -85,B 0,C 180,E1 -19512.806,E2 -19512.806} C_VEL
LIN {X 0,Y 235.149,Z 541.518,A -85,B 0,C 180,E1 -19516.165,E2 -19516.165} C_VEL
LIN {X 0,Y 233.651,Z 542.904,A -85,B 0,C 180,E1 -19519.601,E2 -19519.601} C_VEL
LIN {X 0,Y 233.176,Z 543.028,A -85,B 0,C 180,E1 -19521.331,E2 -19521.331} C_VEL
LIN {X 0,Y 232.922,Z 542.059,A -85,B 0,C 180,E1 -19524.805,E2 -19524.805} C_VEL
LIN {X 0,Y 232.935,Z 542.049,A -85,B 0,C 180,E1 -19525.408,E2 -19525.408} C_VEL
LIN {X 0,Y 232.95,Z 543.292,A -85,B 0,C 180,E1 -19528.269,E2 -19528.269} C_VEL
LIN {X 0,Y 233.063,Z 543.515,A -85,B 0,C 180,E1 -19529.998,E2 -19529.998} C_VEL
LIN {X 0,Y 232.982,Z 543.283,A -85,B 0,C 180,E1 -19531.727,E2 -19531.727} C_VEL
LIN {X 0,Y 232.798,Z 541.621,A -85,B 0,C 180,E1 -19535.194,E2 -19535.194} C_VEL
LIN {X 0,Y 232.882,Z 540.168,A -85,B 0,C 180,E1 -19536.931,E2 -19536.931} C_VEL
LIN {X 0,Y 233.237,Z 537.159,A -85,B 0,C 180,E1 -19539.538,E2 -19539.538} C_VEL
LIN {X 0,Y 233.885,Z 533.084,A -85,B 0,C 180,E1 -19542.141,E2 -19542.141} C_VEL
LIN {X 0,Y 235.359,Z 526.819,A -85,B 0,C 180,E1 -19545.144,E2 -19545.144} C_VEL
LIN {X 0,Y 237.105,Z 519.996,A -85,B 0,C 180,E1 -19547.685,E2 -19547.685} C_VEL
LIN {X 0,Y 238.817,Z 512.822,A -85,B 0,C 180,E1 -19549.841,E2 -19549.841} C_VEL
LIN {X 0,Y 240.74,Z 504.615,A -85,B 0,C 180,E1 -19551.85,E2 -19551.85} C_VEL
LIN {X 0,Y 243.149,Z 494.211,A -85,B 0,C 180,E1 -19553.868,E2 -19553.868} C_VEL
LIN {X 0,Y 245.714,Z 482.503,A -85,B 0,C 180,E1 -19555.631,E2 -19555.631} C_VEL
LIN {X 0,Y 247.732,Z 470.685,A -85,B 0,C 180,E1 -19556.993,E2 -19556.993} C_VEL
LIN {X 0,Y 249.533,Z 458.432,A -85,B 0,C 180,E1 -19558.032,E2 -19558.032} C_VEL
LIN {X 0,Y 250.934,Z 445.753,A -85,B 0,C 180,E1 -19558.774,E2 -19558.774} C_VEL
LIN {X 0,Y 251.761,Z 431.571,A -85,B 0,C 180,E1 -19559.272,E2 -19559.272} C_VEL
LIN {X 0,Y 253.205,Z 386.167,A -85,B 0,C 180,E1 -19560.536,E2 -19560.536} C_VEL
LIN {X 0,Y 249.099,Z 351.41,A -85,B 0,C 180,E1 -19562.237,E2 -19562.237} C_VEL
LIN {X 0,Y 248.178,Z 347.546,A -85,B 0,C 180,E1 -19562.499,E2 -19562.499} C_VEL
LIN {X 0,Y 240.702,Z 326.913,A -85,B 0,C 180,E1 -19564.353,E2 -19564.353} C_VEL
LIN {X 0,Y 236.072,Z 319.188,A -85,B 0,C 180,E1 -19565.405,E2 -19565.405} C_VEL
LIN {X 0,Y 234.981,Z 316.216,A -85,B 0,C 180,E1 -19565.804,E2 -19565.804} C_VEL
LIN {X 0,Y 234.938,Z 316.218,A -85,B 0,C 180,E1 -19568.943,E2 -19568.943} C_VEL
LIN {X 0,Y 234.872,Z 316.22,A -85,B 0,C 180,E1 -19573.487,E2 -19573.487} C_VEL
LIN {X 0,Y 234.857,Z 316.22,A -85,B 0,C 180,E1 -19576.507,E2 -19576.507} C_VEL
LIN {X 0,Y 234.911,Z 316.212,A -85,B 0,C 180,E1 -19581.077,E2 -19581.077} C_VEL
LIN {X 0,Y 234.915,Z 316.214,A -85,B 0,C 180,E1 -19585.359,E2 -19585.359} C_VEL
LIN {X 0,Y 234.887,Z 316.22,A -85,B 0,C 180,E1 -19589.426,E2 -19589.426} C_VEL
LIN {X 0,Y 234.932,Z 316.214,A -85,B 0,C 180,E1 -19593.82,E2 -19593.82} C_VEL
LIN {X 0,Y 234.933,Z 316.216,A -85,B 0,C 180,E1 -19598.962,E2 -19598.962} C_VEL
LIN {X 0,Y 235.047,Z 316.17,A -85,B 0,C 180,E1 -19603.093,E2 -19603.093} C_VEL
LIN {X 0,Y 235.101,Z 316.198,A -85,B 0,C 180,E1 -19607.921,E2 -19607.921} C_VEL
LIN {X 0,Y 235.302,Z 316.157,A -85,B 0,C 180,E1 -19611.411,E2 -19611.411} C_VEL
LIN {X 0,Y 235.339,Z 316.132,A -85,B 0,C 180,E1 -19613.139,E2 -19613.139} C_VEL
LIN {X 0,Y 235.568,Z 316.134,A -85,B 0,C 180,E1 -19618.29,E2 -19618.29} C_VEL
LIN {X 0,Y 235.568,Z 316.136,A -85,B 0,C 180,E1 -19621.71,E2 -19621.71} C_VEL
LIN {X 0,Y 235.338,Z 316.171,A -85,B 0,C 180,E1 -19626.861,E2 -19626.861} C_VEL
LIN {X 0,Y 235.204,Z 316.177,A -85,B 0,C 180,E1 -19630.328,E2 -19630.328} C_VEL
LIN {X 0,Y 235.071,Z 316.192,A -85,B 0,C 180,E1 -19635.609,E2 -19635.609} C_VEL
LIN {X 0,Y 234.98,Z 316.209,A -85,B 0,C 180,E1 -19639.208,E2 -19639.208} C_VEL
LIN {X 0,Y 234.942,Z 316.214,A -85,B 0,C 180,E1 -19642.885,E2 -19642.885} C_VEL
LIN {X 0,Y 234.94,Z 316.212,A -85,B 0,C 180,E1 -19646.661,E2 -19646.661} C_VEL
LIN {X 0,Y 234.893,Z 316.217,A -85,B 0,C 180,E1 -19650.574,E2 -19650.574} C_VEL
LIN {X 0,Y 234.924,Z 316.222,A -85,B 0,C 180,E1 -19654.639,E2 -19654.639} C_VEL
LIN {X 0,Y 234.936,Z 316.213,A -85,B 0,C 180,E1 -19658.946,E2 -19658.946} C_VEL
LIN {X 0,Y 234.875,Z 316.219,A -85,B 0,C 180,E1 -19663.489,E2 -19663.489} C_VEL
LIN {X 0,Y 234.881,Z 316.223,A -85,B 0,C 180,E1 -19666.515,E2 -19666.515} C_VEL
LIN {X 0,Y 234.915,Z 316.211,A -85,B 0,C 180,E1 -19671.081,E2 -19671.081} C_VEL
LIN {X 0,Y 234.951,Z 316.211,A -85,B 0,C 180,E1 -19674.712,E2 -19674.712} C_VEL
LIN {X 0,Y 236.043,Z 319.222,A -85,B 0,C 180,E1 -19675.037,E2 -19675.037} C_VEL
LIN {X 0,Y 237.287,Z 320.98,A -85,B 0,C 180,E1 -19675.313,E2 -19675.313} C_VEL
LIN {X 0,Y 246.992,Z 338.2,A -85,B 0,C 180,E1 -19677.456,E2 -19677.456} C_VEL
LIN {X 0,Y 254.216,Z 353.104,A -85,B 0,C 180,E1 -19678.984,E2 -19678.984} C_VEL
LIN {X 0,Y 254.875,Z 354.56,A -85,B 0,C 180,E1 -19679.121,E2 -19679.121} C_VEL
LIN {X 0,Y 252.425,Z 420.674,A -85,B 0,C 180,E1 -19680.984,E2 -19680.984} C_VEL
LIN {X 0,Y 251.45,Z 433.286,A -85,B 0,C 180,E1 -19681.633,E2 -19681.633} C_VEL
LIN {X 0,Y 250.053,Z 445.792,A -85,B 0,C 180,E1 -19682.6,E2 -19682.6} C_VEL
LIN {X 0,Y 248.4,Z 457.008,A -85,B 0,C 180,E1 -19683.765,E2 -19683.765} C_VEL
LIN {X 0,Y 246.503,Z 467.32,A -85,B 0,C 180,E1 -19685.134,E2 -19685.134} C_VEL
LIN {X 0,Y 244.679,Z 476.567,A -85,B 0,C 180,E1 -19686.681,E2 -19686.681} C_VEL
LIN {X 0,Y 242.479,Z 486.509,A -85,B 0,C 180,E1 -19688.76,E2 -19688.76} C_VEL
LIN {X 0,Y 239.986,Z 495.882,A -85,B 0,C 180,E1 -19691.21,E2 -19691.21} C_VEL
LIN {X 0,Y 238.049,Z 503.317,A -85,B 0,C 180,E1 -19693.713,E2 -19693.713} C_VEL
LIN {X 0,Y 236.372,Z 509.289,A -85,B 0,C 180,E1 -19696.241,E2 -19696.241} C_VEL
LIN {X 0,Y 235.069,Z 514.004,A -85,B 0,C 180,E1 -19698.796,E2 -19698.796} C_VEL
LIN {X 0,Y 234.165,Z 517.602,A -85,B 0,C 180,E1 -19701.371,E2 -19701.371} C_VEL
LIN {X 0,Y 233.71,Z 519.455,A -85,B 0,C 180,E1 -19703.093,E2 -19703.093} C_VEL
LIN {X 0,Y 233.406,Z 520.865,A -85,B 0,C 180,E1 -19704.819,E2 -19704.819} C_VEL
LIN {X 0,Y 233.19,Z 521.854,A -85,B 0,C 180,E1 -19706.546,E2 -19706.546} C_VEL
LIN {X 0,Y 232.96,Z 522.697,A -85,B 0,C 180,E1 -19710.002,E2 -19710.002} C_VEL
LIN {X 0,Y 233.189,Z 521.913,A -85,B 0,C 180,E1 -19713.457,E2 -19713.457} C_VEL
LIN {X 0,Y 233.404,Z 520.947,A -85,B 0,C 180,E1 -19715.184,E2 -19715.184} C_VEL
LIN {X 0,Y 233.819,Z 519.193,A -85,B 0,C 180,E1 -19717.297,E2 -19717.297} C_VEL
LIN {X 0,Y 234.66,Z 515.513,A -85,B 0,C 180,E1 -19720.354,E2 -19720.354} C_VEL
LIN {X 0,Y 235.83,Z 511.241,A -85,B 0,C 180,E1 -19722.917,E2 -19722.917} C_VEL
LIN {X 0,Y 237.376,Z 505.783,A -85,B 0,C 180,E1 -19725.456,E2 -19725.456} C_VEL
LIN {X 0,Y 239.217,Z 498.93,A -85,B 0,C 180,E1 -19727.969,E2 -19727.969} C_VEL
LIN {X 0,Y 241.602,Z 490.331,A -85,B 0,C 180,E1 -19730.432,E2 -19730.432} C_VEL
LIN {X 0,Y 243.674,Z 481.68,A -85,B 0,C 180,E1 -19732.432,E2 -19732.432} C_VEL
LIN {X 0,Y 245.709,Z 471.82,A -85,B 0,C 180,E1 -19734.28,E2 -19734.28} C_VEL
LIN {X 0,Y 247.791,Z 461.056,A -85,B 0,C 180,E1 -19735.855,E2 -19735.855} C_VEL
LIN {X 0,Y 249.694,Z 449.064,A -85,B 0,C 180,E1 -19737.22,E2 -19737.22} C_VEL
LIN {X 0,Y 251.079,Z 437.771,A -85,B 0,C 180,E1 -19738.189,E2 -19738.189} C_VEL
LIN {X 0,Y 252.249,Z 425.02,A -85,B 0,C 180,E1 -19738.945,E2 -19738.945} C_VEL
LIN {X 0,Y 252.997,Z 410.114,A -85,B 0,C 180,E1 -19739.474,E2 -19739.474} C_VEL
LIN {X 0,Y 254.928,Z 354.655,A -85,B 0,C 180,E1 -19741.006,E2 -19741.006} C_VEL
LIN {X 0,Y 247.553,Z 339.164,A -85,B 0,C 180,E1 -19742.569,E2 -19742.569} C_VEL
LIN {X 0,Y 238.59,Z 323.288,A -85,B 0,C 180,E1 -19744.533,E2 -19744.533} C_VEL
LIN {X 0,Y 236.52,Z 319.796,A -85,B 0,C 180,E1 -19745.008,E2 -19745.008} C_VEL
LIN {X 0,Y 235.275,Z 317.5,A -85,B 0,C 180,E1 -19745.307,E2 -19745.307} C_VEL
LIN {X 0,Y 234.999,Z 316.216,A -85,B 0,C 180,E1 -19745.427,E2 -19745.427} C_VEL
LIN {X 0,Y 234.947,Z 316.222,A -85,B 0,C 180,E1 -19748.945,E2 -19748.945} C_VEL
LIN {X 0,Y 234.927,Z 316.213,A -85,B 0,C 180,E1 -19753.479,E2 -19753.479} C_VEL
LIN {X 0,Y 234.896,Z 316.192,A -85,B 0,C 180,E1 -19756.516,E2 -19756.516} C_VEL
LIN {X 0,Y 234.924,Z 316.223,A -85,B 0,C 180,E1 -19761.08,E2 -19761.08} C_VEL
LIN {X 0,Y 234.932,Z 316.22,A -85,B 0,C 180,E1 -19765.362,E2 -19765.362} C_VEL
LIN {X 0,Y 234.937,Z 316.207,A -85,B 0,C 180,E1 -19769.433,E2 -19769.433} C_VEL
LIN {X 0,Y 235.058,Z 316.201,A -85,B 0,C 180,E1 -19774.214,E2 -19774.214} C_VEL
LIN {X 0,Y 242.305,Z 343.599,A -85,B 0,C 180,E1 -19775.906,E2 -19775.906} C_VEL
LIN {X 0,Y 239.024,Z 421.278,A -85,B 0,C 180,E1 -19779.772,E2 -19779.772} C_VEL
LIN {X 0,Y 238.332,Z 433.736,A -85,B 0,C 180,E1 -19780.674,E2 -19780.674} C_VEL
LIN {X 0,Y 237.556,Z 446.51,A -85,B 0,C 180,E1 -19781.902,E2 -19781.902} C_VEL
LIN {X 0,Y 236.662,Z 460.036,A -85,B 0,C 180,E1 -19783.613,E2 -19783.613} C_VEL
LIN {X 0,Y 235.697,Z 470.815,A -85,B 0,C 180,E1 -19785.318,E2 -19785.318} C_VEL
LIN {X 0,Y 234.767,Z 481.819,A -85,B 0,C 180,E1 -19787.465,E2 -19787.465} C_VEL
LIN {X 0,Y 234.093,Z 490.922,A -85,B 0,C 180,E1 -19789.622,E2 -19789.622} C_VEL
LIN {X 0,Y 233.491,Z 499.789,A -85,B 0,C 180,E1 -19792.215,E2 -19792.215} C_VEL
LIN {X 0,Y 233.447,Z 500.811,A -85,B 0,C 180,E1 -19792.552,E2 -19792.552} C_VEL
LIN {X 0,Y 232.641,Z 504.167,A -85,B 0,C 180,E1 -19793.731,E2 -19793.731} C_VEL
LIN {X 0,Y 229.566,Z 508.971,A -85,B 0,C 180,E1 -19795.745,E2 -19795.745} C_VEL
LIN {X 0,Y 226.544,Z 513.12,A -85,B 0,C 180,E1 -19797.905,E2 -19797.905} C_VEL
LIN {X 0,Y 225.847,Z 515.464,A -85,B 0,C 180,E1 -19799.284,E2 -19799.284} C_VEL
LIN {X 0,Y 225.987,Z 519.22,A -85,B 0,C 180,E1 -19801.782,E2 -19801.782} C_VEL
LIN {X 0,Y 226.234,Z 521.354,A -85,B 0,C 180,E1 -19803.562,E2 -19803.562} C_VEL
LIN {X 0,Y 226.513,Z 523.034,A -85,B 0,C 180,E1 -19805.341,E2 -19805.341} C_VEL
LIN {X 0,Y 227.63,Z 525.177,A -85,B 0,C 180,E1 -19808.88,E2 -19808.88} C_VEL
LIN {X 0,Y 229.785,Z 525.777,A -85,B 0,C 180,E1 -19812.362,E2 -19812.362} C_VEL
LIN {X 0,Y 232.525,Z 524.791,A -85,B 0,C 180,E1 -19815.785,E2 -19815.785} C_VEL
LIN {X 0,Y 236.303,Z 522.266,A -85,B 0,C 180,E1 -19819.096,E2 -19819.096} C_VEL
LIN {X 0,Y 239.682,Z 519.282,A -85,B 0,C 180,E1 -19821.502,E2 -19821.502} C_VEL
LIN {X 0,Y 243.492,Z 515.34,A -85,B 0,C 180,E1 -19823.834,E2 -19823.834} C_VEL
LIN {X 0,Y 247.811,Z 510.337,A -85,B 0,C 180,E1 -19826.077,E2 -19826.077} C_VEL
LIN {X 0,Y 253.409,Z 503.021,A -85,B 0,C 180,E1 -19828.581,E2 -19828.581} C_VEL
LIN {X 0,Y 258.671,Z 495.239,A -85,B 0,C 180,E1 -19830.626,E2 -19830.626} C_VEL
LIN {X 0,Y 264.309,Z 485.867,A -85,B 0,C 180,E1 -19832.578,E2 -19832.578} C_VEL
LIN {X 0,Y 269.831,Z 475.362,A -85,B 0,C 180,E1 -19834.28,E2 -19834.28} C_VEL
LIN {X 0,Y 275.123,Z 463.832,A -85,B 0,C 180,E1 -19835.757,E2 -19835.757} C_VEL
LIN {X 0,Y 279.522,Z 452.548,A -85,B 0,C 180,E1 -19836.891,E2 -19836.891} C_VEL
LIN {X 0,Y 283.857,Z 439.348,A -85,B 0,C 180,E1 -19837.903,E2 -19837.903} C_VEL
LIN {X 0,Y 287.133,Z 426.679,A -85,B 0,C 180,E1 -19838.628,E2 -19838.628} C_VEL
LIN {X 0,Y 292.614,Z 402.012,A -85,B 0,C 180,E1 -19839.772,E2 -19839.772} C_VEL
LIN {X 0,Y 292.018,Z 400.701,A -85,B 0,C 180,E1 -19840.836,E2 -19840.836} C_VEL
LIN {X 0,Y 291.14,Z 399.404,A -85,B 0,C 180,E1 -19843.208,E2 -19843.208} C_VEL
LIN {X 0,Y 290.943,Z 399.738,A -85,B 0,C 180,E1 -19845.178,E2 -19845.178} C_VEL
LIN {X 0,Y 291.175,Z 403.254,A -85,B 0,C 180,E1 -19847.86,E2 -19847.86} C_VEL
LIN {X 0,Y 291.459,Z 404.97,A -85,B 0,C 180,E1 -19848.766,E2 -19848.766} C_VEL
LIN {X 0,Y 291.794,Z 407.431,A -85,B 0,C 180,E1 -19849.735,E2 -19849.735} C_VEL
LIN {X 0,Y 284.414,Z 440.207,A -85,B 0,C 180,E1 -19851.24,E2 -19851.24} C_VEL
LIN {X 0,Y 279.485,Z 456.1,A -85,B 0,C 180,E1 -19852.196,E2 -19852.196} C_VEL
LIN {X 0,Y 274.497,Z 469.039,A -85,B 0,C 180,E1 -19853.238,E2 -19853.238} C_VEL
LIN {X 0,Y 269.182,Z 480.91,A -85,B 0,C 180,E1 -19854.455,E2 -19854.455} C_VEL
LIN {X 0,Y 263.628,Z 491.92,A -85,B 0,C 180,E1 -19855.954,E2 -19855.954} C_VEL
LIN {X 0,Y 258.431,Z 501.143,A -85,B 0,C 180,E1 -19857.513,E2 -19857.513} C_VEL
LIN {X 0,Y 252.679,Z 510.462,A -85,B 0,C 180,E1 -19859.494,E2 -19859.494} C_VEL
LIN {X 0,Y 246.719,Z 519.319,A -85,B 0,C 180,E1 -19861.963,E2 -19861.963} C_VEL
LIN {X 0,Y 242.152,Z 525.563,A -85,B 0,C 180,E1 -19864.191,E2 -19864.191} C_VEL
LIN {X 0,Y 238.036,Z 530.719,A -85,B 0,C 180,E1 -19866.508,E2 -19866.508} C_VEL
LIN {X 0,Y 233.748,Z 536.016,A -85,B 0,C 180,E1 -19869.77,E2 -19869.77} C_VEL
LIN {X 0,Y 231.005,Z 538.921,A -85,B 0,C 180,E1 -19872.286,E2 -19872.286} C_VEL
LIN {X 0,Y 228.235,Z 541.485,A -85,B 0,C 180,E1 -19875.737,E2 -19875.737} C_VEL
LIN {X 0,Y 226.644,Z 542.506,A -85,B 0,C 180,E1 -19879.276,E2 -19879.276} C_VEL
LIN {X 0,Y 225.92,Z 542.031,A -85,B 0,C 180,E1 -19882.85,E2 -19882.85} C_VEL
LIN {X 0,Y 225.883,Z 541.336,A -85,B 0,C 180,E1 -19884.642,E2 -19884.642} C_VEL
LIN {X 0,Y 225.857,Z 542.975,A -85,B 0,C 180,E1 -19888.215,E2 -19888.215} C_VEL
LIN {X 0,Y 225.986,Z 543.199,A -85,B 0,C 180,E1 -19889.998,E2 -19889.998} C_VEL
LIN {X 0,Y 225.904,Z 542.967,A -85,B 0,C 180,E1 -19891.781,E2 -19891.781} C_VEL
LIN {X 0,Y 225.728,Z 541.304,A -85,B 0,C 180,E1 -19895.358,E2 -19895.358} C_VEL
LIN {X 0,Y 225.809,Z 539.849,A -85,B 0,C 180,E1 -19897.15,E2 -19897.15} C_VEL
LIN {X 0,Y 226.209,Z 536.84,A -85,B 0,C 180,E1 -19899.837,E2 -19899.837} C_VEL
LIN {X 0,Y 226.896,Z 532.764,A -85,B 0,C 180,E1 -19902.521,E2 -19902.521} C_VEL
LIN {X 0,Y 228.499,Z 526.502,A -85,B 0,C 180,E1 -19905.61,E2 -19905.61} C_VEL
LIN {X 0,Y 230.335,Z 519.68,A -85,B 0,C 180,E1 -19908.223,E2 -19908.223} C_VEL
LIN {X 0,Y 232.393,Z 511.304,A -85,B 0,C 180,E1 -19910.766,E2 -19910.766} C_VEL
LIN {X 0,Y 234.607,Z 502.367,A -85,B 0,C 180,E1 -19912.917,E2 -19912.917} C_VEL
LIN {X 0,Y 236.979,Z 492.738,A -85,B 0,C 180,E1 -19914.763,E2 -19914.763} C_VEL
LIN {X 0,Y 239.331,Z 482.195,A -85,B 0,C 180,E1 -19916.367,E2 -19916.367} C_VEL
LIN {X 0,Y 241.417,Z 470.382,A -85,B 0,C 180,E1 -19917.759,E2 -19917.759} C_VEL
LIN {X 0,Y 243.291,Z 458.137,A -85,B 0,C 180,E1 -19918.818,E2 -19918.818} C_VEL
LIN {X 0,Y 244.719,Z 445.659,A -85,B 0,C 180,E1 -19919.566,E2 -19919.566} C_VEL
LIN {X 0,Y 245.604,Z 430.857,A -85,B 0,C 180,E1 -19920.097,E2 -19920.097} C_VEL
LIN {X 0,Y 247.103,Z 387.416,A -85,B 0,C 180,E1 -19921.326,E2 -19921.326} C_VEL
LIN {X 0,Y 244.012,Z 359.986,A -85,B 0,C 180,E1 -19922.694,E2 -19922.694} C_VEL
LIN {X 0,Y 242.755,Z 351.076,A -85,B 0,C 180,E1 -19923.189,E2 -19923.189} C_VEL
LIN {X 0,Y 235.461,Z 330.727,A -85,B 0,C 180,E1 -19925.084,E2 -19925.084} C_VEL
LIN {X 0,Y 229.674,Z 320.945,A -85,B 0,C 180,E1 -19926.465,E2 -19926.465} C_VEL
LIN {X 0,Y 228.127,Z 318.201,A -85,B 0,C 180,E1 -19926.873,E2 -19926.873} C_VEL
LIN {X 0,Y 227.887,Z 317.093,A -85,B 0,C 180,E1 -19927.027,E2 -19927.027} C_VEL
LIN {X 0,Y 227.82,Z 317.101,A -85,B 0,C 180,E1 -19930.375,E2 -19930.375} C_VEL
LIN {X 0,Y 227.815,Z 317.104,A -85,B 0,C 180,E1 -19935.195,E2 -19935.195} C_VEL
LIN {X 0,Y 227.792,Z 317.104,A -85,B 0,C 180,E1 -19939.616,E2 -19939.616} C_VEL
LIN {X 0,Y 227.855,Z 317.094,A -85,B 0,C 180,E1 -19944.123,E2 -19944.123} C_VEL
LIN {X 0,Y 227.847,Z 317.099,A -85,B 0,C 180,E1 -19948.374,E2 -19948.374} C_VEL
LIN {X 0,Y 227.834,Z 317.104,A -85,B 0,C 180,E1 -19952.438,E2 -19952.438} C_VEL
LIN {X 0,Y 227.859,Z 317.101,A -85,B 0,C 180,E1 -19956.361,E2 -19956.361} C_VEL
LIN {X 0,Y 227.888,Z 317.082,A -85,B 0,C 180,E1 -19960.17,E2 -19960.17} C_VEL
LIN {X 0,Y 228.01,Z 317.051,A -85,B 0,C 180,E1 -19963.894,E2 -19963.894} C_VEL
LIN {X 0,Y 228.056,Z 317.077,A -85,B 0,C 180,E1 -19967.542,E2 -19967.542} C_VEL
LIN {X 0,Y 228.244,Z 317.037,A -85,B 0,C 180,E1 -19971.144,E2 -19971.144} C_VEL
LIN {X 0,Y 228.291,Z 317.01,A -85,B 0,C 180,E1 -19972.927,E2 -19972.927} C_VEL
LIN {X 0,Y 228.526,Z 317.01,A -85,B 0,C 180,E1 -19978.238,E2 -19978.238} C_VEL
LIN {X 0,Y 228.526,Z 317.013,A -85,B 0,C 180,E1 -19981.762,E2 -19981.762} C_VEL
LIN {X 0,Y 228.291,Z 317.048,A -85,B 0,C 180,E1 -19987.074,E2 -19987.074} C_VEL
LIN {X 0,Y 228.134,Z 317.059,A -85,B 0,C 180,E1 -19990.652,E2 -19990.652} C_VEL
LIN {X 0,Y 228.03,Z 317.079,A -85,B 0,C 180,E1 -19994.274,E2 -19994.274} C_VEL
LIN {X 0,Y 227.946,Z 317.075,A -85,B 0,C 180,E1 -19997.958,E2 -19997.958} C_VEL
LIN {X 0,Y 227.914,Z 317.094,A -85,B 0,C 180,E1 -20002.325,E2 -20002.325} C_VEL
LIN {X 0,Y 227.916,Z 317.085,A -85,B 0,C 180,E1 -20006.594,E2 -20006.594} C_VEL
LIN {X 0,Y 227.868,Z 317.095,A -85,B 0,C 180,E1 -20010.282,E2 -20010.282} C_VEL
LIN {X 0,Y 227.871,Z 317.096,A -85,B 0,C 180,E1 -20013.722,E2 -20013.722} C_VEL
LIN {X 0,Y 227.838,Z 317.092,A -85,B 0,C 180,E1 -20018.092,E2 -20018.092} C_VEL
LIN {X 0,Y 227.802,Z 317.1,A -85,B 0,C 180,E1 -20022.745,E2 -20022.745} C_VEL
LIN {X 0,Y 227.806,Z 317.1,A -85,B 0,C 180,E1 -20027.259,E2 -20027.259} C_VEL
LIN {X 0,Y 227.841,Z 317.081,A -85,B 0,C 180,E1 -20031.911,E2 -20031.911} C_VEL
LIN {X 0,Y 227.885,Z 317.075,A -85,B 0,C 180,E1 -20033.477,E2 -20033.477} C_VEL
LIN {X 0,Y 228.887,Z 319.883,A -85,B 0,C 180,E1 -20033.79,E2 -20033.79} C_VEL
LIN {X 0,Y 230.493,Z 322.222,A -85,B 0,C 180,E1 -20034.172,E2 -20034.172} C_VEL
LIN {X 0,Y 240.202,Z 339.085,A -85,B 0,C 180,E1 -20036.439,E2 -20036.439} C_VEL
LIN {X 0,Y 247.928,Z 354.743,A -85,B 0,C 180,E1 -20038.153,E2 -20038.153} C_VEL
LIN {X 0,Y 248.818,Z 356.78,A -85,B 0,C 180,E1 -20038.349,E2 -20038.349} C_VEL
LIN {X 0,Y 246.288,Z 420.547,A -85,B 0,C 180,E1 -20040.172,E2 -20040.172} C_VEL
LIN {X 0,Y 245.247,Z 433.575,A -85,B 0,C 180,E1 -20040.848,E2 -20040.848} C_VEL
LIN {X 0,Y 243.79,Z 446.09,A -85,B 0,C 180,E1 -20041.834,E2 -20041.834} C_VEL
LIN {X 0,Y 242.076,Z 457.313,A -85,B 0,C 180,E1 -20043.025,E2 -20043.025} C_VEL
LIN {X 0,Y 240.08,Z 467.629,A -85,B 0,C 180,E1 -20044.421,E2 -20044.421} C_VEL
LIN {X 0,Y 237.863,Z 478.267,A -85,B 0,C 180,E1 -20046.279,E2 -20046.279} C_VEL
LIN {X 0,Y 235.431,Z 488.557,A -85,B 0,C 180,E1 -20048.552,E2 -20048.552} C_VEL
LIN {X 0,Y 233.299,Z 496.196,A -85,B 0,C 180,E1 -20050.65,E2 -20050.65} C_VEL
LIN {X 0,Y 231.256,Z 503.633,A -85,B 0,C 180,E1 -20053.221,E2 -20053.221} C_VEL
LIN {X 0,Y 229.474,Z 509.606,A -85,B 0,C 180,E1 -20055.819,E2 -20055.819} C_VEL
LIN {X 0,Y 228.107,Z 514.321,A -85,B 0,C 180,E1 -20058.449,E2 -20058.449} C_VEL
LIN {X 0,Y 227.152,Z 517.919,A -85,B 0,C 180,E1 -20061.103,E2 -20061.103} C_VEL
LIN {X 0,Y 226.686,Z 519.771,A -85,B 0,C 180,E1 -20062.878,E2 -20062.878} C_VEL
LIN {X 0,Y 226.35,Z 521.182,A -85,B 0,C 180,E1 -20064.657,E2 -20064.657} C_VEL
LIN {X 0,Y 226.112,Z 522.171,A -85,B 0,C 180,E1 -20066.438,E2 -20066.438} C_VEL
LIN {X 0,Y 225.891,Z 523.013,A -85,B 0,C 180,E1 -20070.002,E2 -20070.002} C_VEL
LIN {X 0,Y 225.941,Z 522.817,A -85,B 0,C 180,E1 -20071.784,E2 -20071.784} C_VEL
LIN {X 0,Y 226.111,Z 522.229,A -85,B 0,C 180,E1 -20073.566,E2 -20073.566} C_VEL
LIN {X 0,Y 226.348,Z 521.263,A -85,B 0,C 180,E1 -20075.347,E2 -20075.347} C_VEL
LIN {X 0,Y 226.738,Z 519.723,A -85,B 0,C 180,E1 -20077.305,E2 -20077.305} C_VEL
LIN {X 0,Y 227.68,Z 515.828,A -85,B 0,C 180,E1 -20080.675,E2 -20080.675} C_VEL
LIN {X 0,Y 228.919,Z 511.556,A -85,B 0,C 180,E1 -20083.314,E2 -20083.314} C_VEL
LIN {X 0,Y 230.558,Z 506.096,A -85,B 0,C 180,E1 -20085.925,E2 -20085.925} C_VEL
LIN {X 0,Y 232.481,Z 499.241,A -85,B 0,C 180,E1 -20088.509,E2 -20088.509} C_VEL
LIN {X 0,Y 234.974,Z 490.639,A -85,B 0,C 180,E1 -20091.035,E2 -20091.035} C_VEL
LIN {X 0,Y 237.03,Z 482.435,A -85,B 0,C 180,E1 -20092.987,E2 -20092.987} C_VEL
LIN {X 0,Y 238.992,Z 473.291,A -85,B 0,C 180,E1 -20094.776,E2 -20094.776} C_VEL
LIN {X 0,Y 241.163,Z 462.877,A -85,B 0,C 180,E1 -20096.388,E2 -20096.388} C_VEL
LIN {X 0,Y 243.151,Z 451.257,A -85,B 0,C 180,E1 -20097.781,E2 -20097.781} C_VEL
LIN {X 0,Y 244.696,Z 439.296,A -85,B 0,C 180,E1 -20098.875,E2 -20098.875} C_VEL
LIN {X 0,Y 245.965,Z 426.634,A -85,B 0,C 180,E1 -20099.68,E2 -20099.68} C_VEL
LIN {X 0,Y 246.81,Z 411.821,A -85,B 0,C 180,E1 -20100.238,E2 -20100.238} C_VEL
LIN {X 0,Y 248.831,Z 356.672,A -85,B 0,C 180,E1 -20101.792,E2 -20101.792} C_VEL
LIN {X 0,Y 241.734,Z 341.985,A -85,B 0,C 180,E1 -20103.361,E2 -20103.361} C_VEL
LIN {X 0,Y 233.572,Z 327.434,A -85,B 0,C 180,E1 -20105.236,E2 -20105.236} C_VEL
LIN {X 0,Y 229.667,Z 320.923,A -85,B 0,C 180,E1 -20106.18,E2 -20106.18} C_VEL
LIN {X 0,Y 228.217,Z 318.382,A -85,B 0,C 180,E1 -20106.546,E2 -20106.546} C_VEL
LIN {X 0,Y 227.91,Z 317.093,A -85,B 0,C 180,E1 -20106.701,E2 -20106.701} C_VEL
LIN {X 0,Y 227.843,Z 317.105,A -85,B 0,C 180,E1 -20110.375,E2 -20110.375} C_VEL
LIN {X 0,Y 227.843,Z 317.073,A -85,B 0,C 180,E1 -20114.809,E2 -20114.809} C_VEL
LIN {X 0,Y 227.832,Z 317.104,A -85,B 0,C 180,E1 -20119.624,E2 -20119.624} C_VEL
LIN {X 0,Y 227.885,Z 317.09,A -85,B 0,C 180,E1 -20124.129,E2 -20124.129} C_VEL
LIN {X 0,Y 227.876,Z 317.09,A -85,B 0,C 180,E1 -20128.379,E2 -20128.379} C_VEL
LIN {X 0,Y 227.894,Z 317.098,A -85,B 0,C 180,E1 -20132.446,E2 -20132.446} C_VEL
LIN {X 0,Y 227.983,Z 317.084,A -85,B 0,C 180,E1 -20133.958,E2 -20133.958} C_VEL
LIN {X 0,Y 235.286,Z 345.312,A -85,B 0,C 180,E1 -20135.751,E2 -20135.751} C_VEL
LIN {X 0,Y 231.908,Z 421.739,A -85,B 0,C 180,E1 -20139.72,E2 -20139.72} C_VEL
LIN {X 0,Y 231.206,Z 434.641,A -85,B 0,C 180,E1 -20140.7,E2 -20140.7} C_VEL
LIN {X 0,Y 230.39,Z 447.608,A -85,B 0,C 180,E1 -20142.016,E2 -20142.016} C_VEL
LIN {X 0,Y 229.43,Z 460.911,A -85,B 0,C 180,E1 -20143.768,E2 -20143.768} C_VEL
LIN {X 0,Y 228.406,Z 472.727,A -85,B 0,C 180,E1 -20145.75,E2 -20145.75} C_VEL
LIN {X 0,Y 227.545,Z 483.467,A -85,B 0,C 180,E1 -20147.966,E2 -20147.966} C_VEL
LIN {X 0,Y 226.916,Z 492.306,A -85,B 0,C 180,E1 -20150.192,E2 -20150.192} C_VEL
LIN {X 0,Y 226.358,Z 500.962,A -85,B 0,C 180,E1 -20152.866,E2 -20152.866} C_VEL
LIN {X 0,Y 226.031,Z 507.984,A -85,B 0,C 180,E1 -20155.542,E2 -20155.542} C_VEL
LIN {X 0,Y 225.898,Z 513.61,A -85,B 0,C 180,E1 -20158.217,E2 -20158.217} C_VEL
LIN {X 0,Y 225.847,Z 515.464,A -85,B 0,C 180,E1 -20159.284,E2 -20159.284} C_VEL
LIN {X 0,Y 225.207,Z 517.624,A -85,B 0,C 180,E1 -20160.675,E2 -20160.675} C_VEL
LIN {X 0,Y 222.536,Z 520.473,A -85,B 0,C 180,E1 -20163.008,E2 -20163.008} C_VEL
LIN {X 0,Y 220.431,Z 522.36,A -85,B 0,C 180,E1 -20164.944,E2 -20164.944} C_VEL
LIN {X 0,Y 219.743,Z 523.615,A -85,B 0,C 180,E1 -20166.449,E2 -20166.449} C_VEL
LIN {X 0,Y 219.799,Z 523.97,A -85,B 0,C 180,E1 -20166.955,E2 -20166.955} C_VEL
LIN {X 0,Y 220.632,Z 525.337,A -85,B 0,C 180,E1 -20169.164,E2 -20169.164} C_VEL
LIN {X 0,Y 222.881,Z 526.242,A -85,B 0,C 180,E1 -20172.752,E2 -20172.752} C_VEL
LIN {X 0,Y 225.767,Z 525.669,A -85,B 0,C 180,E1 -20176.27,E2 -20176.27} C_VEL
LIN {X 0,Y 227.62,Z 524.799,A -85,B 0,C 180,E1 -20177.984,E2 -20177.984} C_VEL
LIN {X 0,Y 232.012,Z 521.849,A -85,B 0,C 180,E1 -20181.315,E2 -20181.315} C_VEL
LIN {X 0,Y 235.862,Z 518.593,A -85,B 0,C 180,E1 -20183.72,E2 -20183.72} C_VEL
LIN {X 0,Y 240.183,Z 514.36,A -85,B 0,C 180,E1 -20186.035,E2 -20186.035} C_VEL
LIN {X 0,Y 245.879,Z 508.031,A -85,B 0,C 180,E1 -20188.605,E2 -20188.605} C_VEL
LIN {X 0,Y 252.089,Z 500.062,A -85,B 0,C 180,E1 -20191.048,E2 -20191.048} C_VEL
LIN {X 0,Y 257.902,Z 491.628,A -85,B 0,C 180,E1 -20193.026,E2 -20193.026} C_VEL
LIN {X 0,Y 264.069,Z 481.437,A -85,B 0,C 180,E1 -20194.904,E2 -20194.904} C_VEL
LIN {X 0,Y 270.086,Z 469.988,A -85,B 0,C 180,E1 -20196.53,E2 -20196.53} C_VEL
LIN {X 0,Y 275.188,Z 458.623,A -85,B 0,C 180,E1 -20197.802,E2 -20197.802} C_VEL
LIN {X 0,Y 279.962,Z 446.101,A -85,B 0,C 180,E1 -20198.872,E2 -20198.872} C_VEL
LIN {X 0,Y 284.261,Z 432.005,A -85,B 0,C 180,E1 -20199.772,E2 -20199.772} C_VEL
LIN {X 0,Y 290.127,Z 407.526,A -85,B 0,C 180,E1 -20200.899,E2 -20200.899} C_VEL
LIN {X 0,Y 289.295,Z 406.257,A -85,B 0,C 180,E1 -20203.212,E2 -20203.212} C_VEL
LIN {X 0,Y 289.089,Z 406.527,A -85,B 0,C 180,E1 -20204.99,E2 -20204.99} C_VEL
LIN {X 0,Y 289.278,Z 410.423,A -85,B 0,C 180,E1 -20207.914,E2 -20207.914} C_VEL
LIN {X 0,Y 289.374,Z 411.883,A -85,B 0,C 180,E1 -20208.537,E2 -20208.537} C_VEL
LIN {X 0,Y 282.945,Z 438.818,A -85,B 0,C 180,E1 -20209.772,E2 -20209.772} C_VEL
LIN {X 0,Y 278.931,Z 451.623,A -85,B 0,C 180,E1 -20210.489,E2 -20210.489} C_VEL
LIN {X 0,Y 273.664,Z 465.291,A -85,B 0,C 180,E1 -20211.48,E2 -20211.48} C_VEL
LIN {X 0,Y 267.278,Z 479.009,A -85,B 0,C 180,E1 -20212.786,E2 -20212.786} C_VEL
LIN {X 0,Y 260.977,Z 490.843,A -85,B 0,C 180,E1 -20214.324,E2 -20214.324} C_VEL
LIN {X 0,Y 254.844,Z 501.081,A -85,B 0,C 180,E1 -20216.05,E2 -20216.05} C_VEL
LIN {X 0,Y 248.757,Z 510.25,A -85,B 0,C 180,E1 -20218.011,E2 -20218.011} C_VEL
LIN {X 0,Y 242.359,Z 518.982,A -85,B 0,C 180,E1 -20220.462,E2 -20220.462} C_VEL
LIN {X 0,Y 237.45,Z 525.144,A -85,B 0,C 180,E1 -20222.691,E2 -20222.691} C_VEL
LIN {X 0,Y 232.97,Z 530.247,A -85,B 0,C 180,E1 -20225.016,E2 -20225.016} C_VEL
LIN {X 0,Y 229.261,Z 534.339,A -85,B 0,C 180,E1 -20227.467,E2 -20227.467} C_VEL
LIN {X 0,Y 226.122,Z 537.538,A -85,B 0,C 180,E1 -20230.006,E2 -20230.006} C_VEL
LIN {X 0,Y 222.657,Z 540.434,A -85,B 0,C 180,E1 -20233.494,E2 -20233.494} C_VEL
LIN {X 0,Y 220.393,Z 541.875,A -85,B 0,C 180,E1 -20237.1,E2 -20237.1} C_VEL
LIN {X 0,Y 219.167,Z 541.858,A -85,B 0,C 180,E1 -20240.772,E2 -20240.772} C_VEL
LIN {X 0,Y 218.839,Z 540.706,A -85,B 0,C 180,E1 -20244.007,E2 -20244.007} C_VEL
LIN {X 0,Y 218.709,Z 542.034,A -85,B 0,C 180,E1 -20246.313,E2 -20246.313} C_VEL
LIN {X 0,Y 218.765,Z 542.658,A -85,B 0,C 180,E1 -20248.157,E2 -20248.157} C_VEL
LIN {X 0,Y 218.911,Z 542.883,A -85,B 0,C 180,E1 -20249.998,E2 -20249.998} C_VEL
LIN {X 0,Y 218.803,Z 542.649,A -85,B 0,C 180,E1 -20251.839,E2 -20251.839} C_VEL
LIN {X 0,Y 218.643,Z 540.985,A -85,B 0,C 180,E1 -20255.532,E2 -20255.532} C_VEL
LIN {X 0,Y 218.725,Z 539.53,A -85,B 0,C 180,E1 -20257.383,E2 -20257.383} C_VEL
LIN {X 0,Y 219.163,Z 536.52,A -85,B 0,C 180,E1 -20260.157,E2 -20260.157} C_VEL
LIN {X 0,Y 219.924,Z 532.445,A -85,B 0,C 180,E1 -20262.924,E2 -20262.924} C_VEL
LIN {X 0,Y 221.65,Z 526.184,A -85,B 0,C 180,E1 -20266.106,E2 -20266.106} C_VEL
LIN {X 0,Y 223.546,Z 519.45,A -85,B 0,C 180,E1 -20268.763,E2 -20268.763} C_VEL
LIN {X 0,Y 225.728,Z 510.988,A -85,B 0,C 180,E1 -20271.409,E2 -20271.409} C_VEL
LIN {X 0,Y 228.073,Z 502.053,A -85,B 0,C 180,E1 -20273.613,E2 -20273.613} C_VEL
LIN {X 0,Y 230.527,Z 492.426,A -85,B 0,C 180,E1 -20275.505,E2 -20275.505} C_VEL
LIN {X 0,Y 232.97,Z 481.886,A -85,B 0,C 180,E1 -20277.145,E2 -20277.145} C_VEL
LIN {X 0,Y 235.163,Z 470.079,A -85,B 0,C 180,E1 -20278.564,E2 -20278.564} C_VEL
LIN {X 0,Y 237.09,Z 457.843,A -85,B 0,C 180,E1 -20279.645,E2 -20279.645} C_VEL
LIN {X 0,Y 238.65,Z 444.81,A -85,B 0,C 180,E1 -20280.429,E2 -20280.429} C_VEL
LIN {X 0,Y 239.495,Z 430.25,A -85,B 0,C 180,E1 -20280.96,E2 -20280.96} C_VEL
LIN {X 0,Y 240.98,Z 387.824,A -85,B 0,C 180,E1 -20282.194,E2 -20282.194} C_VEL
LIN {X 0,Y 237.766,Z 358.784,A -85,B 0,C 180,E1 -20283.7,E2 -20283.7} C_VEL
LIN {X 0,Y 236.903,Z 353.172,A -85,B 0,C 180,E1 -20284.037,E2 -20284.037} C_VEL
LIN {X 0,Y 230.319,Z 334.656,A -85,B 0,C 180,E1 -20285.833,E2 -20285.833} C_VEL
LIN {X 0,Y 224.928,Z 325.525,A -85,B 0,C 180,E1 -20287.178,E2 -20287.178} C_VEL
LIN {X 0,Y 222.741,Z 322.023,A -85,B 0,C 180,E1 -20287.741,E2 -20287.741} C_VEL
LIN {X 0,Y 221.155,Z 319.489,A -85,B 0,C 180,E1 -20288.159,E2 -20288.159} C_VEL
LIN {X 0,Y 220.805,Z 317.981,A -85,B 0,C 180,E1 -20288.347,E2 -20288.347} C_VEL
LIN {X 0,Y 220.756,Z 317.978,A -85,B 0,C 180,E1 -20292.926,E2 -20292.926} C_VEL
LIN {X 0,Y 220.742,Z 317.977,A -85,B 0,C 180,E1 -20297.074,E2 -20297.074} C_VEL
LIN {X 0,Y 220.774,Z 317.972,A -85,B 0,C 180,E1 -20300.456,E2 -20300.456} C_VEL
LIN {X 0,Y 220.818,Z 317.975,A -85,B 0,C 180,E1 -20302.792,E2 -20302.792} C_VEL
LIN {X 0,Y 220.804,Z 317.979,A -85,B 0,C 180,E1 -20307.242,E2 -20307.242} C_VEL
LIN {X 0,Y 220.788,Z 317.982,A -85,B 0,C 180,E1 -20311.48,E2 -20311.48} C_VEL
LIN {X 0,Y 220.796,Z 317.976,A -85,B 0,C 180,E1 -20315.557,E2 -20315.557} C_VEL
LIN {X 0,Y 220.844,Z 317.963,A -85,B 0,C 180,E1 -20319.509,E2 -20319.509} C_VEL
LIN {X 0,Y 220.968,Z 317.921,A -85,B 0,C 180,E1 -20323.366,E2 -20323.366} C_VEL
LIN {X 0,Y 220.993,Z 317.953,A -85,B 0,C 180,E1 -20327.137,E2 -20327.137} C_VEL
LIN {X 0,Y 221.185,Z 317.919,A -85,B 0,C 180,E1 -20330.859,E2 -20330.859} C_VEL
LIN {X 0,Y 221.229,Z 317.89,A -85,B 0,C 180,E1 -20332.7,E2 -20332.7} C_VEL
LIN {X 0,Y 221.46,Z 317.89,A -85,B 0,C 180,E1 -20338.181,E2 -20338.181} C_VEL
LIN {X 0,Y 221.459,Z 317.893,A -85,B 0,C 180,E1 -20341.819,E2 -20341.819} C_VEL
LIN {X 0,Y 221.229,Z 317.926,A -85,B 0,C 180,E1 -20347.301,E2 -20347.301} C_VEL
LIN {X 0,Y 221.054,Z 317.943,A -85,B 0,C 180,E1 -20350.997,E2 -20350.997} C_VEL
LIN {X 0,Y 220.972,Z 317.94,A -85,B 0,C 180,E1 -20356.633,E2 -20356.633} C_VEL
LIN {X 0,Y 220.87,Z 317.971,A -85,B 0,C 180,E1 -20360.488,E2 -20360.488} C_VEL
LIN {X 0,Y 220.843,Z 317.959,A -85,B 0,C 180,E1 -20364.438,E2 -20364.438} C_VEL
LIN {X 0,Y 220.799,Z 317.982,A -85,B 0,C 180,E1 -20368.519,E2 -20368.519} C_VEL
LIN {X 0,Y 220.806,Z 317.967,A -85,B 0,C 180,E1 -20372.758,E2 -20372.758} C_VEL
LIN {X 0,Y 220.805,Z 317.969,A -85,B 0,C 180,E1 -20377.28,E2 -20377.28} C_VEL
LIN {X 0,Y 220.789,Z 317.981,A -85,B 0,C 180,E1 -20380.19,E2 -20380.19} C_VEL
LIN {X 0,Y 220.765,Z 317.981,A -85,B 0,C 180,E1 -20384.457,E2 -20384.457} C_VEL
LIN {X 0,Y 220.765,Z 317.978,A -85,B 0,C 180,E1 -20388.049,E2 -20388.049} C_VEL
LIN {X 0,Y 220.801,Z 318.005,A -85,B 0,C 180,E1 -20392.149,E2 -20392.149} C_VEL
LIN {X 0,Y 221.831,Z 320.827,A -85,B 0,C 180,E1 -20392.47,E2 -20392.47} C_VEL
LIN {X 0,Y 223.565,Z 323.26,A -85,B 0,C 180,E1 -20392.91,E2 -20392.91} C_VEL
LIN {X 0,Y 231.482,Z 336.585,A -85,B 0,C 180,E1 -20394.889,E2 -20394.889} C_VEL
LIN {X 0,Y 238.689,Z 350.158,A -85,B 0,C 180,E1 -20396.59,E2 -20396.59} C_VEL
LIN {X 0,Y 242.679,Z 358.63,A -85,B 0,C 180,E1 -20397.507,E2 -20397.507} C_VEL
LIN {X 0,Y 240.134,Z 421.601,A -85,B 0,C 180,E1 -20399.363,E2 -20399.363} C_VEL
LIN {X 0,Y 239.006,Z 434.578,A -85,B 0,C 180,E1 -20400.07,E2 -20400.07} C_VEL
LIN {X 0,Y 237.424,Z 447.466,A -85,B 0,C 180,E1 -20401.129,E2 -20401.129} C_VEL
LIN {X 0,Y 235.509,Z 459.254,A -85,B 0,C 180,E1 -20402.451,E2 -20402.451} C_VEL
LIN {X 0,Y 233.168,Z 470.466,A -85,B 0,C 180,E1 -20404.086,E2 -20404.086} C_VEL
LIN {X 0,Y 230.793,Z 481.191,A -85,B 0,C 180,E1 -20406.108,E2 -20406.108} C_VEL
LIN {X 0,Y 228.388,Z 490.499,A -85,B 0,C 180,E1 -20408.332,E2 -20408.332} C_VEL
LIN {X 0,Y 225.834,Z 499.164,A -85,B 0,C 180,E1 -20410.93,E2 -20410.93} C_VEL
LIN {X 0,Y 223.802,Z 506.116,A -85,B 0,C 180,E1 -20413.585,E2 -20413.585} C_VEL
LIN {X 0,Y 222.08,Z 511.641,A -85,B 0,C 180,E1 -20416.272,E2 -20416.272} C_VEL
LIN {X 0,Y 220.774,Z 515.966,A -85,B 0,C 180,E1 -20418.991,E2 -20418.991} C_VEL
LIN {X 0,Y 220.136,Z 518.237,A -85,B 0,C 180,E1 -20420.817,E2 -20420.817} C_VEL
LIN {X 0,Y 219.607,Z 520.218,A -85,B 0,C 180,E1 -20422.787,E2 -20422.787} C_VEL
LIN {X 0,Y 219.038,Z 522.488,A -85,B 0,C 180,E1 -20426.323,E2 -20426.323} C_VEL
LIN {X 0,Y 218.823,Z 523.329,A -85,B 0,C 180,E1 -20430.002,E2 -20430.002} C_VEL
LIN {X 0,Y 218.877,Z 523.132,A -85,B 0,C 180,E1 -20431.842,E2 -20431.842} C_VEL
LIN {X 0,Y 219.297,Z 521.579,A -85,B 0,C 180,E1 -20435.519,E2 -20435.519} C_VEL
LIN {X 0,Y 219.645,Z 520.214,A -85,B 0,C 180,E1 -20437.355,E2 -20437.355} C_VEL
LIN {X 0,Y 220.383,Z 517.347,A -85,B 0,C 180,E1 -20440.103,E2 -20440.103} C_VEL
LIN {X 0,Y 221.531,Z 513.441,A -85,B 0,C 180,E1 -20442.833,E2 -20442.833} C_VEL
LIN {X 0,Y 223.119,Z 508.377,A -85,B 0,C 180,E1 -20445.532,E2 -20445.532} C_VEL
LIN {X 0,Y 225.007,Z 501.993,A -85,B 0,C 180,E1 -20448.202,E2 -20448.202} C_VEL
LIN {X 0,Y 227.473,Z 494.034,A -85,B 0,C 180,E1 -20450.814,E2 -20450.814} C_VEL
LIN {X 0,Y 229.788,Z 485.887,A -85,B 0,C 180,E1 -20452.953,E2 -20452.953} C_VEL
LIN {X 0,Y 231.598,Z 477.851,A -85,B 0,C 180,E1 -20454.711,E2 -20454.711} C_VEL
LIN {X 0,Y 233.933,Z 467.346,A -85,B 0,C 180,E1 -20456.546,E2 -20456.546} C_VEL
LIN {X 0,Y 236.348,Z 455.183,A -85,B 0,C 180,E1 -20458.17,E2 -20458.17} C_VEL
LIN {X 0,Y 237.94,Z 444.38,A -85,B 0,C 180,E1 -20459.29,E2 -20459.29} C_VEL
LIN {X 0,Y 239.418,Z 431.659,A -85,B 0,C 180,E1 -20460.244,E2 -20460.244} C_VEL
LIN {X 0,Y 240.416,Z 418.698,A -85,B 0,C 180,E1 -20460.872,E2 -20460.872} C_VEL
LIN {X 0,Y 242.752,Z 358.72,A -85,B 0,C 180,E1 -20462.621,E2 -20462.621} C_VEL
LIN {X 0,Y 235.619,Z 344.055,A -85,B 0,C 180,E1 -20464.277,E2 -20464.277} C_VEL
LIN {X 0,Y 227.111,Z 329.008,A -85,B 0,C 180,E1 -20466.343,E2 -20466.343} C_VEL
LIN {X 0,Y 222.734,Z 321.997,A -85,B 0,C 180,E1 -20467.461,E2 -20467.461} C_VEL
LIN {X 0,Y 221.2,Z 319.495,A -85,B 0,C 180,E1 -20467.869,E2 -20467.869} C_VEL
LIN {X 0,Y 220.83,Z 317.984,A -85,B 0,C 180,E1 -20468.038,E2 -20468.038} C_VEL
LIN {X 0,Y 220.835,Z 317.973,A -85,B 0,C 180,E1 -20472.948,E2 -20472.948} C_VEL
LIN {X 0,Y 220.776,Z 317.964,A -85,B 0,C 180,E1 -20478.049,E2 -20478.049} C_VEL
LIN {X 0,Y 220.812,Z 317.981,A -85,B 0,C 180,E1 -20480.464,E2 -20480.464} C_VEL
LIN {X 0,Y 220.806,Z 317.976,A -85,B 0,C 180,E1 -20485.046,E2 -20485.046} C_VEL
LIN {X 0,Y 220.874,Z 317.958,A -85,B 0,C 180,E1 -20489.396,E2 -20489.396} C_VEL
LIN {X 0,Y 220.93,Z 317.962,A -85,B 0,C 180,E1 -20493.737,E2 -20493.737} C_VEL
LIN {X 0,Y 228.234,Z 346.243,A -85,B 0,C 180,E1 -20495.564,E2 -20495.564} C_VEL
LIN {X 0,Y 224.806,Z 422.453,A -85,B 0,C 180,E1 -20499.702,E2 -20499.702} C_VEL
LIN {X 0,Y 223.952,Z 437.005,A -85,B 0,C 180,E1 -20500.882,E2 -20500.882} C_VEL
LIN {X 0,Y 223.105,Z 450.262,A -85,B 0,C 180,E1 -20502.35,E2 -20502.35} C_VEL
LIN {X 0,Y 222.223,Z 461.605,A -85,B 0,C 180,E1 -20503.935,E2 -20503.935} C_VEL
LIN {X 0,Y 221.257,Z 473.363,A -85,B 0,C 180,E1 -20505.983,E2 -20505.983} C_VEL
LIN {X 0,Y 220.479,Z 483.017,A -85,B 0,C 180,E1 -20508.042,E2 -20508.042} C_VEL
LIN {X 0,Y 219.856,Z 491.988,A -85,B 0,C 180,E1 -20510.339,E2 -20510.339} C_VEL
LIN {X 0,Y 219.245,Z 501.043,A -85,B 0,C 180,E1 -20513.2,E2 -20513.2} C_VEL
LIN {X 0,Y 218.976,Z 508.919,A -85,B 0,C 180,E1 -20516.32,E2 -20516.32} C_VEL
LIN {X 0,Y 218.781,Z 514.848,A -85,B 0,C 180,E1 -20519.352,E2 -20519.352} C_VEL
LIN {X 0,Y 219.025,Z 519.888,A -85,B 0,C 180,E1 -20522.759,E2 -20522.759} C_VEL
LIN {X 0,Y 219.461,Z 522.819,A -85,B 0,C 180,E1 -20525.513,E2 -20525.513} C_VEL
LIN {X 0,Y 219.799,Z 523.97,A -85,B 0,C 180,E1 -20526.955,E2 -20526.955} C_VEL
LIN {X 0,Y 219.67,Z 525.06,A -85,B 0,C 180,E1 -20528.47,E2 -20528.47} C_VEL
LIN {X 0,Y 218.102,Z 526.318,A -85,B 0,C 180,E1 -20531.014,E2 -20531.014} C_VEL
LIN {X 0,Y 217.052,Z 526.782,A -85,B 0,C 180,E1 -20533.084,E2 -20533.084} C_VEL
LIN {X 0,Y 217.205,Z 526.791,A -85,B 0,C 180,E1 -20534.644,E2 -20534.644} C_VEL
LIN {X 0,Y 217.543,Z 526.724,A -85,B 0,C 180,E1 -20535.156,E2 -20535.156} C_VEL
LIN {X 0,Y 220.95,Z 525.766,A -85,B 0,C 180,E1 -20538.547,E2 -20538.547} C_VEL
LIN {X 0,Y 225.548,Z 523.289,A -85,B 0,C 180,E1 -20541.957,E2 -20541.957} C_VEL
LIN {X 0,Y 229.584,Z 520.368,A -85,B 0,C 180,E1 -20544.41,E2 -20544.41} C_VEL
LIN {X 0,Y 234.09,Z 516.516,A -85,B 0,C 180,E1 -20546.766,E2 -20546.766} C_VEL
LIN {X 0,Y 239.114,Z 511.635,A -85,B 0,C 180,E1 -20549.01,E2 -20549.01} C_VEL
LIN {X 0,Y 245.546,Z 504.52,A -85,B 0,C 180,E1 -20551.49,E2 -20551.49} C_VEL
LIN {X 0,Y 252.526,Z 495.571,A -85,B 0,C 180,E1 -20553.822,E2 -20553.822} C_VEL
LIN {X 0,Y 258.89,Z 486.225,A -85,B 0,C 180,E1 -20555.708,E2 -20555.708} C_VEL
LIN {X 0,Y 265.656,Z 474.787,A -85,B 0,C 180,E1 -20557.479,E2 -20557.479} C_VEL
LIN {X 0,Y 271.571,Z 463.071,A -85,B 0,C 180,E1 -20558.871,E2 -20558.871} C_VEL
LIN {X 0,Y 276.525,Z 451.605,A -85,B 0,C 180,E1 -20559.922,E2 -20559.922} C_VEL
LIN {X 0,Y 281.437,Z 437.618,A -85,B 0,C 180,E1 -20560.909,E2 -20560.909} C_VEL
LIN {X 0,Y 285.515,Z 422.6,A -85,B 0,C 180,E1 -20561.653,E2 -20561.653} C_VEL
LIN {X 0,Y 287.721,Z 413.687,A -85,B 0,C 180,E1 -20562.065,E2 -20562.065} C_VEL
LIN {X 0,Y 287.442,Z 413.112,A -85,B 0,C 180,E1 -20563.205,E2 -20563.205} C_VEL
LIN {X 0,Y 287.211,Z 413.455,A -85,B 0,C 180,E1 -20564.942,E2 -20564.942} C_VEL
LIN {X 0,Y 287.199,Z 416.624,A -85,B 0,C 180,E1 -20567.326,E2 -20567.326} C_VEL
LIN {X 0,Y 281.518,Z 438.915,A -85,B 0,C 180,E1 -20568.34,E2 -20568.34} C_VEL
LIN {X 0,Y 276.647,Z 453.247,A -85,B 0,C 180,E1 -20569.143,E2 -20569.143} C_VEL
LIN {X 0,Y 271.164,Z 466.369,A -85,B 0,C 180,E1 -20570.097,E2 -20570.097} C_VEL
LIN {X 0,Y 264.557,Z 479.657,A -85,B 0,C 180,E1 -20571.369,E2 -20571.369} C_VEL
LIN {X 0,Y 258.365,Z 490.467,A -85,B 0,C 180,E1 -20572.752,E2 -20572.752} C_VEL
LIN {X 0,Y 251.363,Z 501.352,A -85,B 0,C 180,E1 -20574.568,E2 -20574.568} C_VEL
LIN {X 0,Y 245.015,Z 510.191,A -85,B 0,C 180,E1 -20576.482,E2 -20576.482} C_VEL
LIN {X 0,Y 239.141,Z 517.654,A -85,B 0,C 180,E1 -20578.556,E2 -20578.556} C_VEL
LIN {X 0,Y 232.933,Z 524.836,A -85,B 0,C 180,E1 -20581.133,E2 -20581.133} C_VEL
LIN {X 0,Y 228.107,Z 529.857,A -85,B 0,C 180,E1 -20583.463,E2 -20583.463} C_VEL
LIN {X 0,Y 223.91,Z 533.906,A -85,B 0,C 180,E1 -20585.916,E2 -20585.916} C_VEL
LIN {X 0,Y 219.464,Z 537.895,A -85,B 0,C 180,E1 -20589.373,E2 -20589.373} C_VEL
LIN {X 0,Y 215.849,Z 540.441,A -85,B 0,C 180,E1 -20592.958,E2 -20592.958} C_VEL
LIN {X 0,Y 214.457,Z 541.15,A -85,B 0,C 180,E1 -20594.799,E2 -20594.799} C_VEL
LIN {X 0,Y 212.68,Z 541.491,A -85,B 0,C 180,E1 -20598.562,E2 -20598.562} C_VEL
LIN {X 0,Y 211.91,Z 540.393,A -85,B 0,C 180,E1 -20602.375,E2 -20602.375} C_VEL
LIN {X 0,Y 211.836,Z 540.023,A -85,B 0,C 180,E1 -20603.33,E2 -20603.33} C_VEL
LIN {X 0,Y 211.622,Z 541.717,A -85,B 0,C 180,E1 -20606.19,E2 -20606.19} C_VEL
LIN {X 0,Y 211.676,Z 542.342,A -85,B 0,C 180,E1 -20608.095,E2 -20608.095} C_VEL
LIN {X 0,Y 211.837,Z 542.567,A -85,B 0,C 180,E1 -20609.998,E2 -20609.998} C_VEL
LIN {X 0,Y 211.706,Z 542.332,A -85,B 0,C 180,E1 -20611.9,E2 -20611.9} C_VEL
LIN {X 0,Y 211.564,Z 540.667,A -85,B 0,C 180,E1 -20615.718,E2 -20615.718} C_VEL
LIN {X 0,Y 211.653,Z 539.211,A -85,B 0,C 180,E1 -20617.631,E2 -20617.631} C_VEL
LIN {X 0,Y 212.122,Z 536.201,A -85,B 0,C 180,E1 -20620.497,E2 -20620.497} C_VEL
LIN {X 0,Y 212.963,Z 532.126,A -85,B 0,C 180,E1 -20623.354,E2 -20623.354} C_VEL
LIN {X 0,Y 214.799,Z 525.866,A -85,B 0,C 180,E1 -20626.634,E2 -20626.634} C_VEL
LIN {X 0,Y 216.935,Z 518.608,A -85,B 0,C 180,E1 -20629.565,E2 -20629.565} C_VEL
LIN {X 0,Y 219.146,Z 510.509,A -85,B 0,C 180,E1 -20632.135,E2 -20632.135} C_VEL
LIN {X 0,Y 221.557,Z 501.738,A -85,B 0,C 180,E1 -20634.352,E2 -20634.352} C_VEL
LIN {X 0,Y 224.125,Z 492.114,A -85,B 0,C 180,E1 -20636.288,E2 -20636.288} C_VEL
LIN {X 0,Y 226.661,Z 481.577,A -85,B 0,C 180,E1 -20637.966,E2 -20637.966} C_VEL
LIN {X 0,Y 228.958,Z 469.777,A -85,B 0,C 180,E1 -20639.413,E2 -20639.413} C_VEL
LIN {X 0,Y 230.959,Z 457.55,A -85,B 0,C 180,E1 -20640.515,E2 -20640.515} C_VEL
LIN {X 0,Y 232.55,Z 444.759,A -85,B 0,C 180,E1 -20641.303,E2 -20641.303} C_VEL
LIN {X 0,Y 233.453,Z 429.76,A -85,B 0,C 180,E1 -20641.863,E2 -20641.863} C_VEL
LIN {X 0,Y 235.006,Z 388.968,A -85,B 0,C 180,E1 -20643.067,E2 -20643.067} C_VEL
LIN {X 0,Y 231.971,Z 360.854,A -85,B 0,C 180,E1 -20644.576,E2 -20644.576} C_VEL
LIN {X 0,Y 231.163,Z 355.532,A -85,B 0,C 180,E1 -20644.909,E2 -20644.909} C_VEL
LIN {X 0,Y 225.054,Z 338.184,A -85,B 0,C 180,E1 -20646.662,E2 -20646.662} C_VEL
LIN {X 0,Y 218.487,Z 327.158,A -85,B 0,C 180,E1 -20648.393,E2 -20648.393} C_VEL
LIN {X 0,Y 216.325,Z 323.65,A -85,B 0,C 180,E1 -20648.99,E2 -20648.99} C_VEL
LIN {X 0,Y 214.243,Z 320.695,A -85,B 0,C 180,E1 -20649.564,E2 -20649.564} C_VEL
LIN {X 0,Y 213.777,Z 318.849,A -85,B 0,C 180,E1 -20649.782,E2 -20649.782} C_VEL
LIN {X 0,Y 213.698,Z 318.857,A -85,B 0,C 180,E1 -20653.678,E2 -20653.678} C_VEL
LIN {X 0,Y 213.696,Z 318.855,A -85,B 0,C 180,E1 -20656.344,E2 -20656.344} C_VEL
LIN {X 0,Y 213.695,Z 318.855,A -85,B 0,C 180,E1 -20661.327,E2 -20661.327} C_VEL
LIN {X 0,Y 213.746,Z 318.854,A -85,B 0,C 180,E1 -20666.016,E2 -20666.016} C_VEL
LIN {X 0,Y 213.739,Z 318.856,A -85,B 0,C 180,E1 -20670.448,E2 -20670.448} C_VEL
LIN {X 0,Y 213.743,Z 318.85,A -85,B 0,C 180,E1 -20674.694,E2 -20674.694} C_VEL
LIN {X 0,Y 213.771,Z 318.851,A -85,B 0,C 180,E1 -20678.799,E2 -20678.799} C_VEL
LIN {X 0,Y 213.877,Z 318.8,A -85,B 0,C 180,E1 -20682.798,E2 -20682.798} C_VEL
LIN {X 0,Y 213.931,Z 318.83,A -85,B 0,C 180,E1 -20686.705,E2 -20686.705} C_VEL
LIN {X 0,Y 214.125,Z 318.801,A -85,B 0,C 180,E1 -20690.555,E2 -20690.555} C_VEL
LIN {X 0,Y 214.065,Z 318.77,A -85,B 0,C 180,E1 -20694.348,E2 -20694.348} C_VEL
LIN {X 0,Y 214.397,Z 318.769,A -85,B 0,C 180,E1 -20698.122,E2 -20698.122} C_VEL
LIN {X 0,Y 214.502,Z 318.763,A -85,B 0,C 180,E1 -20700,E2 -20700} C_VEL
LIN {X 0,Y 214.395,Z 318.773,A -85,B 0,C 180,E1 -20701.879,E2 -20701.879} C_VEL
LIN {X 0,Y 214.171,Z 318.804,A -85,B 0,C 180,E1 -20707.542,E2 -20707.542} C_VEL
LIN {X 0,Y 213.986,Z 318.826,A -85,B 0,C 180,E1 -20711.365,E2 -20711.365} C_VEL
LIN {X 0,Y 213.894,Z 318.83,A -85,B 0,C 180,E1 -20715.24,E2 -20715.24} C_VEL
LIN {X 0,Y 213.807,Z 318.843,A -85,B 0,C 180,E1 -20719.19,E2 -20719.19} C_VEL
LIN {X 0,Y 213.796,Z 318.844,A -85,B 0,C 180,E1 -20723.233,E2 -20723.233} C_VEL
LIN {X 0,Y 213.782,Z 318.854,A -85,B 0,C 180,E1 -20727.43,E2 -20727.43} C_VEL
LIN {X 0,Y 213.752,Z 318.842,A -85,B 0,C 180,E1 -20731.74,E2 -20731.74} C_VEL
LIN {X 0,Y 213.738,Z 318.856,A -85,B 0,C 180,E1 -20736.29,E2 -20736.29} C_VEL
LIN {X 0,Y 213.706,Z 318.864,A -85,B 0,C 180,E1 -20741.127,E2 -20741.127} C_VEL
LIN {X 0,Y 213.698,Z 318.856,A -85,B 0,C 180,E1 -20743.681,E2 -20743.681} C_VEL
LIN {X 0,Y 213.7,Z 318.861,A -85,B 0,C 180,E1 -20746.346,E2 -20746.346} C_VEL
LIN {X 0,Y 213.756,Z 318.848,A -85,B 0,C 180,E1 -20750.658,E2 -20750.658} C_VEL
LIN {X 0,Y 214.825,Z 321.828,A -85,B 0,C 180,E1 -20751.051,E2 -20751.051} C_VEL
LIN {X 0,Y 216.557,Z 324.147,A -85,B 0,C 180,E1 -20751.521,E2 -20751.521} C_VEL
LIN {X 0,Y 223.535,Z 335.534,A -85,B 0,C 180,E1 -20753.39,E2 -20753.39} C_VEL
LIN {X 0,Y 231.421,Z 349.884,A -85,B 0,C 180,E1 -20755.374,E2 -20755.374} C_VEL
LIN {X 0,Y 236.656,Z 360.7,A -85,B 0,C 180,E1 -20756.64,E2 -20756.64} C_VEL
LIN {X 0,Y 234.087,Z 421.671,A -85,B 0,C 180,E1 -20758.474,E2 -20758.474} C_VEL
LIN {X 0,Y 232.902,Z 434.868,A -85,B 0,C 180,E1 -20759.202,E2 -20759.202} C_VEL
LIN {X 0,Y 231.252,Z 447.766,A -85,B 0,C 180,E1 -20760.283,E2 -20760.283} C_VEL
LIN {X 0,Y 229.256,Z 459.56,A -85,B 0,C 180,E1 -20761.632,E2 -20761.632} C_VEL
LIN {X 0,Y 226.827,Z 470.775,A -85,B 0,C 180,E1 -20763.306,E2 -20763.306} C_VEL
LIN {X 0,Y 224.451,Z 480.874,A -85,B 0,C 180,E1 -20765.238,E2 -20765.238} C_VEL
LIN {X 0,Y 222.311,Z 489.184,A -85,B 0,C 180,E1 -20767.218,E2 -20767.218} C_VEL
LIN {X 0,Y 219.99,Z 496.825,A -85,B 0,C 180,E1 -20769.428,E2 -20769.428} C_VEL
LIN {X 0,Y 217.712,Z 504.265,A -85,B 0,C 180,E1 -20772.143,E2 -20772.143} C_VEL
LIN {X 0,Y 215.751,Z 510.239,A -85,B 0,C 180,E1 -20774.897,E2 -20774.897} C_VEL
LIN {X 0,Y 214.238,Z 514.954,A -85,B 0,C 180,E1 -20777.69,E2 -20777.69} C_VEL
LIN {X 0,Y 213.151,Z 518.553,A -85,B 0,C 180,E1 -20780.513,E2 -20780.513} C_VEL
LIN {X 0,Y 212.514,Z 520.741,A -85,B 0,C 180,E1 -20782.807,E2 -20782.807} C_VEL
LIN {X 0,Y 211.967,Z 522.805,A -85,B 0,C 180,E1 -20786.2,E2 -20786.2} C_VEL
LIN {X 0,Y 211.816,Z 523.414,A -85,B 0,C 180,E1 -20788.101,E2 -20788.101} C_VEL
LIN {X 0,Y 211.757,Z 523.644,A -85,B 0,C 180,E1 -20790.002,E2 -20790.002} C_VEL
LIN {X 0,Y 211.815,Z 523.447,A -85,B 0,C 180,E1 -20791.903,E2 -20791.903} C_VEL
LIN {X 0,Y 212.229,Z 521.896,A -85,B 0,C 180,E1 -20795.703,E2 -20795.703} C_VEL
LIN {X 0,Y 212.621,Z 520.529,A -85,B 0,C 180,E1 -20797.6,E2 -20797.6} C_VEL
LIN {X 0,Y 213.407,Z 517.662,A -85,B 0,C 180,E1 -20800.437,E2 -20800.437} C_VEL
LIN {X 0,Y 214.632,Z 513.755,A -85,B 0,C 180,E1 -20803.252,E2 -20803.252} C_VEL
LIN {X 0,Y 216.29,Z 508.69,A -85,B 0,C 180,E1 -20806.035,E2 -20806.035} C_VEL
LIN {X 0,Y 218.27,Z 502.306,A -85,B 0,C 180,E1 -20808.785,E2 -20808.785} C_VEL
LIN {X 0,Y 220.859,Z 494.344,A -85,B 0,C 180,E1 -20811.468,E2 -20811.468} C_VEL
LIN {X 0,Y 223.275,Z 486.195,A -85,B 0,C 180,E1 -20813.663,E2 -20813.663} C_VEL
LIN {X 0,Y 225.638,Z 476.174,A -85,B 0,C 180,E1 -20815.855,E2 -20815.855} C_VEL
LIN {X 0,Y 228.24,Z 464.888,A -85,B 0,C 180,E1 -20817.759,E2 -20817.759} C_VEL
LIN {X 0,Y 230.416,Z 453.738,A -85,B 0,C 180,E1 -20819.212,E2 -20819.212} C_VEL
LIN {X 0,Y 232.094,Z 442.314,A -85,B 0,C 180,E1 -20820.354,E2 -20820.354} C_VEL
LIN {X 0,Y 233.594,Z 429.372,A -85,B 0,C 180,E1 -20821.269,E2 -20821.269} C_VEL
LIN {X 0,Y 234.512,Z 416.602,A -85,B 0,C 180,E1 -20821.842,E2 -20821.842} C_VEL
LIN {X 0,Y 236.748,Z 360.836,A -85,B 0,C 180,E1 -20823.487,E2 -20823.487} C_VEL
LIN {X 0,Y 229.843,Z 346.774,A -85,B 0,C 180,E1 -20825.169,E2 -20825.169} C_VEL
LIN {X 0,Y 222.075,Z 332.988,A -85,B 0,C 180,E1 -20827.152,E2 -20827.152} C_VEL
LIN {X 0,Y 217.865,Z 326.323,A -85,B 0,C 180,E1 -20828.276,E2 -20828.276} C_VEL
LIN {X 0,Y 215.77,Z 322.979,A -85,B 0,C 180,E1 -20828.86,E2 -20828.86} C_VEL
LIN {X 0,Y 214.137,Z 320.396,A -85,B 0,C 180,E1 -20829.325,E2 -20829.325} C_VEL
LIN {X 0,Y 213.776,Z 318.855,A -85,B 0,C 180,E1 -20829.532,E2 -20829.532} C_VEL
LIN {X 0,Y 213.753,Z 318.839,A -85,B 0,C 180,E1 -20833.669,E2 -20833.669} C_VEL
LIN {X 0,Y 213.718,Z 318.855,A -85,B 0,C 180,E1 -20838.876,E2 -20838.876} C_VEL
LIN {X 0,Y 213.749,Z 318.848,A -85,B 0,C 180,E1 -20843.712,E2 -20843.712} C_VEL
LIN {X 0,Y 213.774,Z 318.846,A -85,B 0,C 180,E1 -20848.263,E2 -20848.263} C_VEL
LIN {X 0,Y 213.883,Z 318.853,A -85,B 0,C 180,E1 -20853.513,E2 -20853.513} C_VEL
LIN {X 0,Y 221.139,Z 346.974,A -85,B 0,C 180,E1 -20855.373,E2 -20855.373} C_VEL
LIN {X 0,Y 217.682,Z 423.271,A -85,B 0,C 180,E1 -20859.716,E2 -20859.716} C_VEL
LIN {X 0,Y 216.84,Z 437.199,A -85,B 0,C 180,E1 -20860.89,E2 -20860.89} C_VEL
LIN {X 0,Y 215.927,Z 450.956,A -85,B 0,C 180,E1 -20862.478,E2 -20862.478} C_VEL
LIN {X 0,Y 215.077,Z 462.188,A -85,B 0,C 180,E1 -20864.117,E2 -20864.117} C_VEL
LIN {X 0,Y 214.127,Z 473.849,A -85,B 0,C 180,E1 -20866.234,E2 -20866.234} C_VEL
LIN {X 0,Y 213.265,Z 484.457,A -85,B 0,C 180,E1 -20868.596,E2 -20868.596} C_VEL
LIN {X 0,Y 212.57,Z 494.718,A -85,B 0,C 180,E1 -20871.444,E2 -20871.444} C_VEL
LIN {X 0,Y 212.074,Z 503.054,A -85,B 0,C 180,E1 -20874.294,E2 -20874.294} C_VEL
LIN {X 0,Y 211.885,Z 509.744,A -85,B 0,C 180,E1 -20877.148,E2 -20877.148} C_VEL
LIN {X 0,Y 211.732,Z 515.105,A -85,B 0,C 180,E1 -20880,E2 -20880} C_VEL
LIN {X 0,Y 211.968,Z 519.329,A -85,B 0,C 180,E1 -20882.851,E2 -20882.851} C_VEL
LIN {X 0,Y 212.413,Z 522.542,A -85,B 0,C 180,E1 -20885.696,E2 -20885.696} C_VEL
LIN {X 0,Y 213.641,Z 525.36,A -85,B 0,C 180,E1 -20889.467,E2 -20889.467} C_VEL
LIN {X 0,Y 215.972,Z 526.677,A -85,B 0,C 180,E1 -20893.167,E2 -20893.167} C_VEL
LIN {X 0,Y 217.543,Z 526.724,A -85,B 0,C 180,E1 -20895.156,E2 -20895.156} C_VEL
LIN {X 0,Y 218.272,Z 526.559,A -85,B 0,C 180,E1 -20896.699,E2 -20896.699} C_VEL
LIN {X 0,Y 218.403,Z 525.325,A -85,B 0,C 180,E1 -20901.369,E2 -20901.369} C_VEL
LIN {X 0,Y 219.531,Z 524.406,A -85,B 0,C 180,E1 -20902.858,E2 -20902.858} C_VEL
LIN {X 0,Y 220.19,Z 523.968,A -85,B 0,C 180,E1 -20903.327,E2 -20903.327} C_VEL
LIN {X 0,Y 224.857,Z 521.003,A -85,B 0,C 180,E1 -20905.949,E2 -20905.949} C_VEL
LIN {X 0,Y 229.717,Z 517.225,A -85,B 0,C 180,E1 -20908.308,E2 -20908.308} C_VEL
LIN {X 0,Y 235.097,Z 512.436,A -85,B 0,C 180,E1 -20910.544,E2 -20910.544} C_VEL
LIN {X 0,Y 241.936,Z 505.464,A -85,B 0,C 180,E1 -20913.002,E2 -20913.002} C_VEL
LIN {X 0,Y 248.238,Z 498.075,A -85,B 0,C 180,E1 -20914.981,E2 -20914.981} C_VEL
LIN {X 0,Y 254.647,Z 489.538,A -85,B 0,C 180,E1 -20916.787,E2 -20916.787} C_VEL
LIN {X 0,Y 261.508,Z 479.146,A -85,B 0,C 180,E1 -20918.495,E2 -20918.495} C_VEL
LIN {X 0,Y 267.45,Z 468.698,A -85,B 0,C 180,E1 -20919.831,E2 -20919.831} C_VEL
LIN {X 0,Y 272.541,Z 458.378,A -85,B 0,C 180,E1 -20920.885,E2 -20920.885} C_VEL
LIN {X 0,Y 278.171,Z 444.733,A -85,B 0,C 180,E1 -20921.94,E2 -20921.94} C_VEL
LIN {X 0,Y 282.283,Z 432.301,A -85,B 0,C 180,E1 -20922.656,E2 -20922.656} C_VEL
LIN {X 0,Y 285.584,Z 419.944,A -85,B 0,C 180,E1 -20923.231,E2 -20923.231} C_VEL
LIN {X 0,Y 285.319,Z 420.398,A -85,B 0,C 180,E1 -20924.847,E2 -20924.847} C_VEL
LIN {X 0,Y 285.158,Z 422.05,A -85,B 0,C 180,E1 -20926.133,E2 -20926.133} C_VEL
LIN {X 0,Y 280.334,Z 439.495,A -85,B 0,C 180,E1 -20926.913,E2 -20926.913} C_VEL
LIN {X 0,Y 275.295,Z 453.411,A -85,B 0,C 180,E1 -20927.673,E2 -20927.673} C_VEL
LIN {X 0,Y 269.585,Z 466.32,A -85,B 0,C 180,E1 -20928.582,E2 -20928.582} C_VEL
LIN {X 0,Y 262.721,Z 479.401,A -85,B 0,C 180,E1 -20929.805,E2 -20929.805} C_VEL
LIN {X 0,Y 255.556,Z 491.079,A -85,B 0,C 180,E1 -20931.269,E2 -20931.269} C_VEL
LIN {X 0,Y 248.299,Z 501.581,A -85,B 0,C 180,E1 -20933.023,E2 -20933.023} C_VEL
LIN {X 0,Y 240.971,Z 510.951,A -85,B 0,C 180,E1 -20935.083,E2 -20935.083} C_VEL
LIN {X 0,Y 234.274,Z 518.707,A -85,B 0,C 180,E1 -20937.316,E2 -20937.316} C_VEL
LIN {X 0,Y 228.618,Z 524.644,A -85,B 0,C 180,E1 -20939.519,E2 -20939.519} C_VEL
LIN {X 0,Y 223.472,Z 529.553,A -85,B 0,C 180,E1 -20941.851,E2 -20941.851} C_VEL
LIN {X 0,Y 218.877,Z 533.526,A -85,B 0,C 180,E1 -20944.31,E2 -20944.31} C_VEL
LIN {X 0,Y 215.068,Z 536.616,A -85,B 0,C 180,E1 -20946.911,E2 -20946.911} C_VEL
LIN {X 0,Y 210.832,Z 539.432,A -85,B 0,C 180,E1 -20950.526,E2 -20950.526} C_VEL
LIN {X 0,Y 207.6,Z 540.851,A -85,B 0,C 180,E1 -20954.285,E2 -20954.285} C_VEL
LIN {X 0,Y 205.723,Z 540.875,A -85,B 0,C 180,E1 -20958.17,E2 -20958.17} C_VEL
LIN {X 0,Y 204.923,Z 539.428,A -85,B 0,C 180,E1 -20962.113,E2 -20962.113} C_VEL
LIN {X 0,Y 204.862,Z 539.34,A -85,B 0,C 180,E1 -20962.607,E2 -20962.607} C_VEL
LIN {X 0,Y 204.54,Z 541.401,A -85,B 0,C 180,E1 -20966.058,E2 -20966.058} C_VEL
LIN {X 0,Y 204.589,Z 542.025,A -85,B 0,C 180,E1 -20968.029,E2 -20968.029} C_VEL
LIN {X 0,Y 204.763,Z 542.251,A -85,B 0,C 180,E1 -20969.998,E2 -20969.998} C_VEL
LIN {X 0,Y 204.611,Z 542.014,A -85,B 0,C 180,E1 -20971.966,E2 -20971.966} C_VEL
LIN {X 0,Y 204.466,Z 541.109,A -85,B 0,C 180,E1 -20974.582,E2 -20974.582} C_VEL
LIN {X 0,Y 204.603,Z 538.893,A -85,B 0,C 180,E1 -20977.895,E2 -20977.895} C_VEL
LIN {X 0,Y 205.102,Z 535.881,A -85,B 0,C 180,E1 -20980.861,E2 -20980.861} C_VEL
LIN {X 0,Y 206.017,Z 531.806,A -85,B 0,C 180,E1 -20983.813,E2 -20983.813} C_VEL
LIN {X 0,Y 207.955,Z 525.547,A -85,B 0,C 180,E1 -20987.198,E2 -20987.198} C_VEL
LIN {X 0,Y 210.112,Z 518.618,A -85,B 0,C 180,E1 -20990.093,E2 -20990.093} C_VEL
LIN {X 0,Y 212.535,Z 510.192,A -85,B 0,C 180,E1 -20992.862,E2 -20992.862} C_VEL
LIN {X 0,Y 215.098,Z 501.425,A -85,B 0,C 180,E1 -20995.133,E2 -20995.133} C_VEL
LIN {X 0,Y 217.762,Z 491.802,A -85,B 0,C 180,E1 -20997.119,E2 -20997.119} C_VEL
LIN {X 0,Y 220.399,Z 481.269,A -85,B 0,C 180,E1 -20998.833,E2 -20998.833} C_VEL
LIN {X 0,Y 222.81,Z 469.476,A -85,B 0,C 180,E1 -21000.308,E2 -21000.308} C_VEL
LIN {X 0,Y 224.874,Z 457.256,A -85,B 0,C 180,E1 -21001.433,E2 -21001.433} C_VEL
LIN {X 0,Y 226.503,Z 444.704,A -85,B 0,C 180,E1 -21002.225,E2 -21002.225} C_VEL
LIN {X 0,Y 227.417,Z 430.54,A -85,B 0,C 180,E1 -21002.776,E2 -21002.776} C_VEL
LIN {X 0,Y 229.056,Z 389.907,A -85,B 0,C 180,E1 -21003.999,E2 -21003.999} C_VEL
LIN {X 0,Y 226.172,Z 362.165,A -85,B 0,C 180,E1 -21005.536,E2 -21005.536} C_VEL
LIN {X 0,Y 225.419,Z 357.679,A -85,B 0,C 180,E1 -21005.844,E2 -21005.844} C_VEL
LIN {X 0,Y 219.965,Z 341.964,A -85,B 0,C 180,E1 -21007.495,E2 -21007.495} C_VEL
LIN {X 0,Y 213.967,Z 331.893,A -85,B 0,C 180,E1 -21009.151,E2 -21009.151} C_VEL
LIN {X 0,Y 209.396,Z 324.597,A -85,B 0,C 180,E1 -21010.488,E2 -21010.488} C_VEL
LIN {X 0,Y 207.278,Z 321.875,A -85,B 0,C 180,E1 -21011.108,E2 -21011.108} C_VEL
LIN {X 0,Y 206.655,Z 319.74,A -85,B 0,C 180,E1 -21011.421,E2 -21011.421} C_VEL
LIN {X 0,Y 206.625,Z 319.74,A -85,B 0,C 180,E1 -21015.581,E2 -21015.581} C_VEL
LIN {X 0,Y 206.64,Z 319.735,A -85,B 0,C 180,E1 -21019.744,E2 -21019.744} C_VEL
LIN {X 0,Y 206.693,Z 319.727,A -85,B 0,C 180,E1 -21024.687,E2 -21024.687} C_VEL
LIN {X 0,Y 206.687,Z 319.731,A -85,B 0,C 180,E1 -21029.333,E2 -21029.333} C_VEL
LIN {X 0,Y 206.678,Z 319.732,A -85,B 0,C 180,E1 -21033.765,E2 -21033.765} C_VEL
LIN {X 0,Y 206.707,Z 319.734,A -85,B 0,C 180,E1 -21038.038,E2 -21038.038} C_VEL
LIN {X 0,Y 206.814,Z 319.678,A -85,B 0,C 180,E1 -21042.191,E2 -21042.191} C_VEL
LIN {X 0,Y 206.871,Z 319.707,A -85,B 0,C 180,E1 -21046.243,E2 -21046.243} C_VEL
LIN {X 0,Y 207.07,Z 319.683,A -85,B 0,C 180,E1 -21050.23,E2 -21050.23} C_VEL
LIN {X 0,Y 207.028,Z 319.644,A -85,B 0,C 180,E1 -21054.155,E2 -21054.155} C_VEL
LIN {X 0,Y 207.336,Z 319.646,A -85,B 0,C 180,E1 -21058.058,E2 -21058.058} C_VEL
LIN {X 0,Y 207.47,Z 319.639,A -85,B 0,C 180,E1 -21060,E2 -21060} C_VEL
LIN {X 0,Y 207.335,Z 319.652,A -85,B 0,C 180,E1 -21061.943,E2 -21061.943} C_VEL
LIN {X 0,Y 207.116,Z 319.682,A -85,B 0,C 180,E1 -21067.801,E2 -21067.801} C_VEL
LIN {X 0,Y 206.909,Z 319.71,A -85,B 0,C 180,E1 -21071.759,E2 -21071.759} C_VEL
LIN {X 0,Y 206.822,Z 319.705,A -85,B 0,C 180,E1 -21075.774,E2 -21075.774} C_VEL
LIN {X 0,Y 206.743,Z 319.729,A -85,B 0,C 180,E1 -21079.873,E2 -21079.873} C_VEL
LIN {X 0,Y 206.732,Z 319.716,A -85,B 0,C 180,E1 -21084.076,E2 -21084.076} C_VEL
LIN {X 0,Y 206.683,Z 319.74,A -85,B 0,C 180,E1 -21088.428,E2 -21088.428} C_VEL
LIN {X 0,Y 206.689,Z 319.725,A -85,B 0,C 180,E1 -21092.96,E2 -21092.96} C_VEL
LIN {X 0,Y 206.674,Z 319.726,A -85,B 0,C 180,E1 -21097.741,E2 -21097.741} C_VEL
LIN {X 0,Y 206.636,Z 319.743,A -85,B 0,C 180,E1 -21101.564,E2 -21101.564} C_VEL
LIN {X 0,Y 206.627,Z 319.747,A -85,B 0,C 180,E1 -21105.584,E2 -21105.584} C_VEL
LIN {X 0,Y 206.669,Z 319.742,A -85,B 0,C 180,E1 -21109.086,E2 -21109.086} C_VEL
LIN {X 0,Y 207.656,Z 322.555,A -85,B 0,C 180,E1 -21109.453,E2 -21109.453} C_VEL
LIN {X 0,Y 209.604,Z 325.087,A -85,B 0,C 180,E1 -21110.023,E2 -21110.023} C_VEL
LIN {X 0,Y 217.192,Z 337.177,A -85,B 0,C 180,E1 -21112.194,E2 -21112.194} C_VEL
LIN {X 0,Y 225.045,Z 351.251,A -85,B 0,C 180,E1 -21114.289,E2 -21114.289} C_VEL
LIN {X 0,Y 230.679,Z 362.932,A -85,B 0,C 180,E1 -21115.731,E2 -21115.731} C_VEL
LIN {X 0,Y 228.087,Z 421.852,A -85,B 0,C 180,E1 -21117.541,E2 -21117.541} C_VEL
LIN {X 0,Y 226.945,Z 434.442,A -85,B 0,C 180,E1 -21118.236,E2 -21118.236} C_VEL
LIN {X 0,Y 225.303,Z 446.988,A -85,B 0,C 180,E1 -21119.286,E2 -21119.286} C_VEL
LIN {X 0,Y 223.347,Z 458.228,A -85,B 0,C 180,E1 -21120.552,E2 -21120.552} C_VEL
LIN {X 0,Y 221.086,Z 468.557,A -85,B 0,C 180,E1 -21122.041,E2 -21122.041} C_VEL
LIN {X 0,Y 218.868,Z 477.979,A -85,B 0,C 180,E1 -21123.774,E2 -21123.774} C_VEL
LIN {X 0,Y 216.304,Z 487.763,A -85,B 0,C 180,E1 -21126.04,E2 -21126.04} C_VEL
LIN {X 0,Y 213.362,Z 497.141,A -85,B 0,C 180,E1 -21128.759,E2 -21128.759} C_VEL
LIN {X 0,Y 210.939,Z 504.583,A -85,B 0,C 180,E1 -21131.55,E2 -21131.55} C_VEL
LIN {X 0,Y 208.919,Z 510.555,A -85,B 0,C 180,E1 -21134.39,E2 -21134.39} C_VEL
LIN {X 0,Y 207.305,Z 515.272,A -85,B 0,C 180,E1 -21137.272,E2 -21137.272} C_VEL
LIN {X 0,Y 206.158,Z 518.871,A -85,B 0,C 180,E1 -21140.188,E2 -21140.188} C_VEL
LIN {X 0,Y 205.442,Z 521.216,A -85,B 0,C 180,E1 -21142.78,E2 -21142.78} C_VEL
LIN {X 0,Y 204.899,Z 523.121,A -85,B 0,C 180,E1 -21146.068,E2 -21146.068} C_VEL
LIN {X 0,Y 204.692,Z 523.96,A -85,B 0,C 180,E1 -21150.002,E2 -21150.002} C_VEL
LIN {X 0,Y 204.732,Z 523.764,A -85,B 0,C 180,E1 -21151.969,E2 -21151.969} C_VEL
LIN {X 0,Y 204.898,Z 523.177,A -85,B 0,C 180,E1 -21153.936,E2 -21153.936} C_VEL
LIN {X 0,Y 205.442,Z 521.321,A -85,B 0,C 180,E1 -21157.22,E2 -21157.22} C_VEL
LIN {X 0,Y 206.433,Z 517.977,A -85,B 0,C 180,E1 -21160.794,E2 -21160.794} C_VEL
LIN {X 0,Y 207.721,Z 514.07,A -85,B 0,C 180,E1 -21163.702,E2 -21163.702} C_VEL
LIN {X 0,Y 209.487,Z 509.003,A -85,B 0,C 180,E1 -21166.571,E2 -21166.571} C_VEL
LIN {X 0,Y 211.561,Z 502.618,A -85,B 0,C 180,E1 -21169.404,E2 -21169.404} C_VEL
LIN {X 0,Y 214.273,Z 494.654,A -85,B 0,C 180,E1 -21172.162,E2 -21172.162} C_VEL
LIN {X 0,Y 216.793,Z 486.503,A -85,B 0,C 180,E1 -21174.416,E2 -21174.416} C_VEL
LIN {X 0,Y 219.003,Z 477.613,A -85,B 0,C 180,E1 -21176.442,E2 -21176.442} C_VEL
LIN {X 0,Y 221.63,Z 466.568,A -85,B 0,C 180,E1 -21178.404,E2 -21178.404} C_VEL
LIN {X 0,Y 223.966,Z 455.768,A -85,B 0,C 180,E1 -21179.88,E2 -21179.88} C_VEL
LIN {X 0,Y 225.672,Z 444.95,A -85,B 0,C 180,E1 -21181.053,E2 -21181.053} C_VEL
LIN {X 0,Y 227.271,Z 432.546,A -85,B 0,C 180,E1 -21182.018,E2 -21182.018} C_VEL
LIN {X 0,Y 228.383,Z 419.103,A -85,B 0,C 180,E1 -21182.696,E2 -21182.696} C_VEL
LIN {X 0,Y 230.791,Z 363.011,A -85,B 0,C 180,E1 -21184.397,E2 -21184.397} C_VEL
LIN {X 0,Y 224.233,Z 349.714,A -85,B 0,C 180,E1 -21186.078,E2 -21186.078} C_VEL
LIN {X 0,Y 216.188,Z 335.366,A -85,B 0,C 180,E1 -21188.252,E2 -21188.252} C_VEL
LIN {X 0,Y 210.774,Z 327.044,A -85,B 0,C 180,E1 -21189.792,E2 -21189.792} C_VEL
LIN {X 0,Y 208.957,Z 324.076,A -85,B 0,C 180,E1 -21190.343,E2 -21190.343} C_VEL
LIN {X 0,Y 207.219,Z 321.657,A -85,B 0,C 180,E1 -21190.863,E2 -21190.863} C_VEL
LIN {X 0,Y 206.7,Z 319.743,A -85,B 0,C 180,E1 -21191.077,E2 -21191.077} C_VEL
LIN {X 0,Y 206.649,Z 319.702,A -85,B 0,C 180,E1 -21195.58,E2 -21195.58} C_VEL
LIN {X 0,Y 206.667,Z 319.741,A -85,B 0,C 180,E1 -21199.75,E2 -21199.75} C_VEL
LIN {X 0,Y 206.705,Z 319.73,A -85,B 0,C 180,E1 -21204.69,E2 -21204.69} C_VEL
LIN {X 0,Y 206.72,Z 319.719,A -85,B 0,C 180,E1 -21209.338,E2 -21209.338} C_VEL
LIN {X 0,Y 206.862,Z 319.836,A -85,B 0,C 180,E1 -21213.283,E2 -21213.283} C_VEL
LIN {X 0,Y 214.064,Z 347.823,A -85,B 0,C 180,E1 -21215.204,E2 -21215.204} C_VEL
LIN {X 0,Y 210.584,Z 423.467,A -85,B 0,C 180,E1 -21219.709,E2 -21219.709} C_VEL
LIN {X 0,Y 209.704,Z 437.366,A -85,B 0,C 180,E1 -21220.928,E2 -21220.928} C_VEL
LIN {X 0,Y 208.785,Z 451.508,A -85,B 0,C 180,E1 -21222.618,E2 -21222.618} C_VEL
LIN {X 0,Y 207.867,Z 462.594,A -85,B 0,C 180,E1 -21224.307,E2 -21224.307} C_VEL
LIN {X 0,Y 206.965,Z 474.203,A -85,B 0,C 180,E1 -21226.499,E2 -21226.499} C_VEL
LIN {X 0,Y 206.206,Z 483.797,A -85,B 0,C 180,E1 -21228.698,E2 -21228.698} C_VEL
LIN {X 0,Y 205.624,Z 492.693,A -85,B 0,C 180,E1 -21231.152,E2 -21231.152} C_VEL
LIN {X 0,Y 205.082,Z 501.385,A -85,B 0,C 180,E1 -21234.099,E2 -21234.099} C_VEL
LIN {X 0,Y 204.881,Z 508.464,A -85,B 0,C 180,E1 -21237.05,E2 -21237.05} C_VEL
LIN {X 0,Y 204.686,Z 514.131,A -85,B 0,C 180,E1 -21240,E2 -21240} C_VEL
LIN {X 0,Y 204.914,Z 518.642,A -85,B 0,C 180,E1 -21242.949,E2 -21242.949} C_VEL
LIN {X 0,Y 205.369,Z 522.115,A -85,B 0,C 180,E1 -21245.893,E2 -21245.893} C_VEL
LIN {X 0,Y 206.644,Z 525.335,A -85,B 0,C 180,E1 -21249.791,E2 -21249.791} C_VEL
LIN {X 0,Y 209.071,Z 526.975,A -85,B 0,C 180,E1 -21253.61,E2 -21253.61} C_VEL
LIN {X 0,Y 212.251,Z 527.152,A -85,B 0,C 180,E1 -21257.338,E2 -21257.338} C_VEL
LIN {X 0,Y 216.593,Z 525.854,A -85,B 0,C 180,E1 -21260.912,E2 -21260.912} C_VEL
LIN {X 0,Y 220.19,Z 523.968,A -85,B 0,C 180,E1 -21263.327,E2 -21263.327} C_VEL
LIN {X 0,Y 221.925,Z 522.752,A -85,B 0,C 180,E1 -21264.758,E2 -21264.758} C_VEL
LIN {X 0,Y 224.211,Z 519.903,A -85,B 0,C 180,E1 -21268.198,E2 -21268.198} C_VEL
LIN {X 0,Y 226.273,Z 517.641,A -85,B 0,C 180,E1 -21270.039,E2 -21270.039} C_VEL
LIN {X 0,Y 227.936,Z 516.178,A -85,B 0,C 180,E1 -21270.852,E2 -21270.852} C_VEL
LIN {X 0,Y 235.378,Z 509.643,A -85,B 0,C 180,E1 -21273.531,E2 -21273.531} C_VEL
LIN {X 0,Y 242.04,Z 502.877,A -85,B 0,C 180,E1 -21275.605,E2 -21275.605} C_VEL
LIN {X 0,Y 249.815,Z 493.75,A -85,B 0,C 180,E1 -21277.726,E2 -21277.726} C_VEL
LIN {X 0,Y 256.955,Z 484.143,A -85,B 0,C 180,E1 -21279.437,E2 -21279.437} C_VEL
LIN {X 0,Y 264.043,Z 473.021,A -85,B 0,C 180,E1 -21280.953,E2 -21280.953} C_VEL
LIN {X 0,Y 269.94,Z 462.297,A -85,B 0,C 180,E1 -21282.099,E2 -21282.099} C_VEL
LIN {X 0,Y 276.059,Z 448.922,A -85,B 0,C 180,E1 -21283.172,E2 -21283.172} C_VEL
LIN {X 0,Y 280.953,Z 435.594,A -85,B 0,C 180,E1 -21283.97,E2 -21283.97} C_VEL
LIN {X 0,Y 283.518,Z 426.998,A -85,B 0,C 180,E1 -21284.361,E2 -21284.361} C_VEL
LIN {X 0,Y 283.398,Z 427.52,A -85,B 0,C 180,E1 -21284.911,E2 -21284.911} C_VEL
LIN {X 0,Y 278.78,Z 442.289,A -85,B 0,C 180,E1 -21285.574,E2 -21285.574} C_VEL
LIN {X 0,Y 273.611,Z 455.359,A -85,B 0,C 180,E1 -21286.291,E2 -21286.291} C_VEL
LIN {X 0,Y 267.554,Z 468.008,A -85,B 0,C 180,E1 -21287.18,E2 -21287.18} C_VEL
LIN {X 0,Y 260.437,Z 480.54,A -85,B 0,C 180,E1 -21288.353,E2 -21288.353} C_VEL
LIN {X 0,Y 252.984,Z 491.899,A -85,B 0,C 180,E1 -21289.765,E2 -21289.765} C_VEL
LIN {X 0,Y 244.154,Z 503.583,A -85,B 0,C 180,E1 -21291.764,E2 -21291.764} C_VEL
LIN {X 0,Y 235.988,Z 513.07,A -85,B 0,C 180,E1 -21293.97,E2 -21293.97} C_VEL
LIN {X 0,Y 228.512,Z 520.791,A -85,B 0,C 180,E1 -21296.384,E2 -21296.384} C_VEL
LIN {X 0,Y 222.677,Z 526.231,A -85,B 0,C 180,E1 -21298.615,E2 -21298.615} C_VEL
LIN {X 0,Y 215.744,Z 531.981,A -85,B 0,C 180,E1 -21301.765,E2 -21301.765} C_VEL
LIN {X 0,Y 211.105,Z 535.31,A -85,B 0,C 180,E1 -21304.353,E2 -21304.353} C_VEL
LIN {X 0,Y 206.23,Z 538.431,A -85,B 0,C 180,E1 -21307.982,E2 -21307.982} C_VEL
LIN {X 0,Y 202.31,Z 540.133,A -85,B 0,C 180,E1 -21311.779,E2 -21311.779} C_VEL
LIN {X 0,Y 199.662,Z 540.459,A -85,B 0,C 180,E1 -21315.734,E2 -21315.734} C_VEL
LIN {X 0,Y 198.243,Z 539.416,A -85,B 0,C 180,E1 -21319.788,E2 -21319.788} C_VEL
LIN {X 0,Y 197.954,Z 538.525,A -85,B 0,C 180,E1 -21321.705,E2 -21321.705} C_VEL
LIN {X 0,Y 197.506,Z 540.749,A -85,B 0,C 180,E1 -21325.1,E2 -21325.1} C_VEL
LIN {X 0,Y 197.505,Z 541.709,A -85,B 0,C 180,E1 -21327.959,E2 -21327.959} C_VEL
LIN {X 0,Y 197.691,Z 541.935,A -85,B 0,C 180,E1 -21329.998,E2 -21329.998} C_VEL
LIN {X 0,Y 197.519,Z 541.697,A -85,B 0,C 180,E1 -21332.037,E2 -21332.037} C_VEL
LIN {X 0,Y 197.371,Z 540.925,A -85,B 0,C 180,E1 -21334.417,E2 -21334.417} C_VEL
LIN {X 0,Y 197.529,Z 538.573,A -85,B 0,C 180,E1 -21338.18,E2 -21338.18} C_VEL
LIN {X 0,Y 198.102,Z 535.562,A -85,B 0,C 180,E1 -21341.25,E2 -21341.25} C_VEL
LIN {X 0,Y 199.091,Z 531.488,A -85,B 0,C 180,E1 -21344.304,E2 -21344.304} C_VEL
LIN {X 0,Y 201.115,Z 525.227,A -85,B 0,C 180,E1 -21347.802,E2 -21347.802} C_VEL
LIN {X 0,Y 203.305,Z 518.626,A -85,B 0,C 180,E1 -21350.656,E2 -21350.656} C_VEL
LIN {X 0,Y 205.517,Z 511.442,A -85,B 0,C 180,E1 -21353.155,E2 -21353.155} C_VEL
LIN {X 0,Y 208.087,Z 503.042,A -85,B 0,C 180,E1 -21355.505,E2 -21355.505} C_VEL
LIN {X 0,Y 211.134,Z 492.653,A -85,B 0,C 180,E1 -21357.774,E2 -21357.774} C_VEL
LIN {X 0,Y 213.823,Z 482.375,A -85,B 0,C 180,E1 -21359.537,E2 -21359.537} C_VEL
LIN {X 0,Y 216.32,Z 471.104,A -85,B 0,C 180,E1 -21361.046,E2 -21361.046} C_VEL
LIN {X 0,Y 218.645,Z 458.227,A -85,B 0,C 180,E1 -21362.3,E2 -21362.3} C_VEL
LIN {X 0,Y 220.434,Z 445.236,A -85,B 0,C 180,E1 -21363.167,E2 -21363.167} C_VEL
LIN {X 0,Y 221.443,Z 431.27,A -85,B 0,C 180,E1 -21363.74,E2 -21363.74} C_VEL
LIN {X 0,Y 223.124,Z 390.016,A -85,B 0,C 180,E1 -21365.02,E2 -21365.02} C_VEL
LIN {X 0,Y 220.162,Z 361.164,A -85,B 0,C 180,E1 -21366.692,E2 -21366.692} C_VEL
LIN {X 0,Y 214.943,Z 345.825,A -85,B 0,C 180,E1 -21368.361,E2 -21368.361} C_VEL
LIN {X 0,Y 209.365,Z 336.421,A -85,B 0,C 180,E1 -21369.978,E2 -21369.978} C_VEL
LIN {X 0,Y 204.436,Z 328.865,A -85,B 0,C 180,E1 -21371.481,E2 -21371.481} C_VEL
LIN {X 0,Y 202.086,Z 325.21,A -85,B 0,C 180,E1 -21372.239,E2 -21372.239} C_VEL
LIN {X 0,Y 200.207,Z 322.777,A -85,B 0,C 180,E1 -21372.841,E2 -21372.841} C_VEL
LIN {X 0,Y 199.582,Z 320.613,A -85,B 0,C 180,E1 -21373.147,E2 -21373.147} C_VEL
LIN {X 0,Y 199.564,Z 320.618,A -85,B 0,C 180,E1 -21378.001,E2 -21378.001} C_VEL
LIN {X 0,Y 199.59,Z 320.61,A -85,B 0,C 180,E1 -21380.771,E2 -21380.771} C_VEL
LIN {X 0,Y 199.603,Z 320.612,A -85,B 0,C 180,E1 -21385.712,E2 -21385.712} C_VEL
LIN {X 0,Y 199.678,Z 320.608,A -85,B 0,C 180,E1 -21388.133,E2 -21388.133} C_VEL
LIN {X 0,Y 199.627,Z 320.618,A -85,B 0,C 180,E1 -21392.763,E2 -21392.763} C_VEL
LIN {X 0,Y 199.664,Z 320.615,A -85,B 0,C 180,E1 -21397.22,E2 -21397.22} C_VEL
LIN {X 0,Y 199.738,Z 320.559,A -85,B 0,C 180,E1 -21401.802,E2 -21401.802} C_VEL
LIN {X 0,Y 199.807,Z 320.579,A -85,B 0,C 180,E1 -21405.746,E2 -21405.746} C_VEL
LIN {X 0,Y 200.015,Z 320.563,A -85,B 0,C 180,E1 -21409.881,E2 -21409.881} C_VEL
LIN {X 0,Y 199.992,Z 320.519,A -85,B 0,C 180,E1 -21413.948,E2 -21413.948} C_VEL
LIN {X 0,Y 200.278,Z 320.522,A -85,B 0,C 180,E1 -21417.989,E2 -21417.989} C_VEL
LIN {X 0,Y 200.438,Z 320.515,A -85,B 0,C 180,E1 -21420,E2 -21420} C_VEL
LIN {X 0,Y 199.976,Z 320.563,A -85,B 0,C 180,E1 -21424.031,E2 -21424.031} C_VEL
LIN {X 0,Y 200.065,Z 320.56,A -85,B 0,C 180,E1 -21428.078,E2 -21428.078} C_VEL
LIN {X 0,Y 199.858,Z 320.588,A -85,B 0,C 180,E1 -21432.18,E2 -21432.18} C_VEL
LIN {X 0,Y 199.759,Z 320.58,A -85,B 0,C 180,E1 -21436.347,E2 -21436.347} C_VEL
LIN {X 0,Y 199.666,Z 320.613,A -85,B 0,C 180,E1 -21440.609,E2 -21440.609} C_VEL
LIN {X 0,Y 199.645,Z 320.595,A -85,B 0,C 180,E1 -21444.988,E2 -21444.988} C_VEL
LIN {X 0,Y 199.603,Z 320.62,A -85,B 0,C 180,E1 -21449.534,E2 -21449.534} C_VEL
LIN {X 0,Y 199.659,Z 320.597,A -85,B 0,C 180,E1 -21452.354,E2 -21452.354} C_VEL
LIN {X 0,Y 199.617,Z 320.61,A -85,B 0,C 180,E1 -21456.765,E2 -21456.765} C_VEL
LIN {X 0,Y 199.602,Z 320.613,A -85,B 0,C 180,E1 -21459.33,E2 -21459.33} C_VEL
LIN {X 0,Y 199.567,Z 320.616,A -85,B 0,C 180,E1 -21462.311,E2 -21462.311} C_VEL
LIN {X 0,Y 199.608,Z 320.79,A -85,B 0,C 180,E1 -21467.345,E2 -21467.345} C_VEL
LIN {X 0,Y 200.694,Z 323.657,A -85,B 0,C 180,E1 -21467.769,E2 -21467.769} C_VEL
LIN {X 0,Y 202.643,Z 326.009,A -85,B 0,C 180,E1 -21468.381,E2 -21468.381} C_VEL
LIN {X 0,Y 204.845,Z 329.321,A -85,B 0,C 180,E1 -21469.082,E2 -21469.082} C_VEL
LIN {X 0,Y 212.839,Z 342.147,A -85,B 0,C 180,E1 -21471.483,E2 -21471.483} C_VEL
LIN {X 0,Y 220.962,Z 357.048,A -85,B 0,C 180,E1 -21473.748,E2 -21473.748} C_VEL
LIN {X 0,Y 224.75,Z 364.956,A -85,B 0,C 180,E1 -21474.764,E2 -21474.764} C_VEL
LIN {X 0,Y 222.138,Z 422.112,A -85,B 0,C 180,E1 -21476.559,E2 -21476.559} C_VEL
LIN {X 0,Y 220.952,Z 434.731,A -85,B 0,C 180,E1 -21477.269,E2 -21477.269} C_VEL
LIN {X 0,Y 219.248,Z 447.286,A -85,B 0,C 180,E1 -21478.341,E2 -21478.341} C_VEL
LIN {X 0,Y 217.208,Z 458.533,A -85,B 0,C 180,E1 -21479.634,E2 -21479.634} C_VEL
LIN {X 0,Y 214.852,Z 468.866,A -85,B 0,C 180,E1 -21481.154,E2 -21481.154} C_VEL
LIN {X 0,Y 212.118,Z 479.757,A -85,B 0,C 180,E1 -21483.247,E2 -21483.247} C_VEL
LIN {X 0,Y 209.327,Z 489.811,A -85,B 0,C 180,E1 -21485.717,E2 -21485.717} C_VEL
LIN {X 0,Y 206.774,Z 497.456,A -85,B 0,C 180,E1 -21488.047,E2 -21488.047} C_VEL
LIN {X 0,Y 204.21,Z 504.9,A -85,B 0,C 180,E1 -21490.919,E2 -21490.919} C_VEL
LIN {X 0,Y 202.09,Z 510.872,A -85,B 0,C 180,E1 -21493.849,E2 -21493.849} C_VEL
LIN {X 0,Y 200.397,Z 515.589,A -85,B 0,C 180,E1 -21496.825,E2 -21496.825} C_VEL
LIN {X 0,Y 199.163,Z 519.188,A -85,B 0,C 180,E1 -21499.84,E2 -21499.84} C_VEL
LIN {X 0,Y 198.315,Z 521.782,A -85,B 0,C 180,E1 -21502.878,E2 -21502.878} C_VEL
LIN {X 0,Y 197.833,Z 523.438,A -85,B 0,C 180,E1 -21505.928,E2 -21505.928} C_VEL
LIN {X 0,Y 197.606,Z 524.276,A -85,B 0,C 180,E1 -21510.002,E2 -21510.002} C_VEL
LIN {X 0,Y 197.652,Z 524.08,A -85,B 0,C 180,E1 -21512.04,E2 -21512.04} C_VEL
LIN {X 0,Y 197.833,Z 523.493,A -85,B 0,C 180,E1 -21514.076,E2 -21514.076} C_VEL
LIN {X 0,Y 198.358,Z 521.815,A -85,B 0,C 180,E1 -21517.22,E2 -21517.22} C_VEL
LIN {X 0,Y 199.46,Z 518.293,A -85,B 0,C 180,E1 -21521.176,E2 -21521.176} C_VEL
LIN {X 0,Y 200.831,Z 514.385,A -85,B 0,C 180,E1 -21524.182,E2 -21524.182} C_VEL
LIN {X 0,Y 202.689,Z 509.317,A -85,B 0,C 180,E1 -21527.143,E2 -21527.143} C_VEL
